// TIA Portal project "Boiler S7 1200+HMI_test_program" (V15)

(* hardware
DEVICE "S7-1200 station_1"  S7-1200 Station
   slot 0: "Rack_0"  S7-1200 Rack  Rack  V1.0
   slot 1: "PLC_BOILER_S71200"  CPU 1214C DC/DC/DC  6ES7 214-1AG40-0XB0  V4.2
   slot 2: "DI 16/DQ 16x24VDC_1"  6ES7 223-1BL32-0XB0  V2.0
   slot 3: "DI 16/DQ 16x24VDC_2"  6ES7 223-1BL32-0XB0  V2.0
   slot 4: "DI 16/DQ 16x24VDC_3"  6ES7 223-1BL32-0XB0  V2.0
   slot 5: "AI 8x13BIT_1"  6ES7 231-4HF32-0XB0  V2.0
   slot 6: "AI 8x13BIT_2"  6ES7 231-4HF32-0XB0  V2.0
   slot 7: "AI 8x13BIT_3"  6ES7 231-4HF32-0XB0  V2.0
   slot 8: "AQ 4x14BIT_1"  6ES7 232-4HD32-0XB0  V2.0
   slot 9: "AQ 4x14BIT_2"  6ES7 232-4HD32-0XB0  V2.0
DEVICE "HMI_BOILER_S71200"  TP1200 Comfort
   slot 0: "HMI_BOILER_S71200"  TP1200 Comfort  6AV2 124-0MC01-0AX0  14.0.1.0
   slot 1: "HMI_RT_2"  TP1200 Comfort  6AV2 124-0MC01-0AX0  14.0.1.0
   slot 5: "HMI_BOILER_S71200.IE_CP_1"  PROFINET Interface  14.0.1.0
      slot 1: "PROFINET Interface_1"  PROFINET Interface
         slot 1: "Port_1"  Port
         slot 2: "Port_2"  Port
   slot 7: "HMI_BOILER_S71200.MPI/DP_CP_1"  MPI/DP Interface  14.0.1.0
*)

// ===== PLC "PLC_BOILER_S71200"  CPU 1214C DC/DC/DC =====

VAR_GLOBAL   // PLC tag table "Default tag table"
   "Tag_2" AT %M4.2 : Bool;
   "Tag_3" AT %M4.3 : Bool;
   "PUMP_COMP_VALUE" AT %MD104 : Real;
   "REFF_PUMPS_FINAL" AT %MD108 : Real;
   "Tag_7" AT %MD128 : Real;
   "Tag_8" AT %MD124 : Real;
   "Tag_9" AT %MD120 : Real;
   "ALRM_Feed_Pump_1_Fault" AT %M15.3 : Bool;
   "ROUND_O2_LEVEL" AT %MD112 : DWord;
   "ROUND SP O2" AT %MD116 : DWord;
   "ID Fan Start" AT %Q0.2 : Bool;
   "Block LH FD Fan" AT %Q4.0 : Bool;
   "Block RH FD Fan" AT %Q4.1 : Bool;
   "Tag_16" AT %M21.5 : Bool;
   "LH_COAL_HEIGHT_0" AT %M13.0 : Bool;
   "RH_COAL_HEIGHT_0" AT %M13.1 : Bool;
   "ALRM_Low_Water_PreWarning" AT %M15.0 : Bool;
   "ALRM_Low_Water" AT %M15.1 : Bool;
   "ALRM_High_Water" AT %M15.2 : Bool;
   "ALRM_Feed_Pump_2_Fault" AT %M15.4 : Bool;
   "ALRM_ID_Fan_Fault" AT %M15.5 : Bool;
   "ALRM_LH_FD_Fan_Fault" AT %M15.6 : Bool;
   "ALRM_RH_FD_Fan_Fault" AT %M15.7 : Bool;
   "ALRM_LH_Stoker_Fault" AT %M14.0 : Bool;
   "ALRM_RH_Stoker_Fault" AT %M14.1 : Bool;
   "ALRM_LH_Swing_Chute_Fault" AT %M14.2 : Bool;
   "ALRM_RH_Swing_Chute_Fault" AT %M14.3 : Bool;
   "ALRM_RAV_1_Fault" AT %M14.4 : Bool;
   "ALRM_RAV_2_Fault" AT %M14.5 : Bool;
   "ALRM_Ash_Conv_Fault" AT %M14.6 : Bool;
   "ALRM_LH_Shearpin_Fault" AT %M14.7 : Bool;
   "ALRM_RH_Shearpin_Fault" AT %M17.0 : Bool;
   "ALRM_LH_Burnback_Fault" AT %M17.1 : Bool;
   "ALRM_RH_Burnback_Fault" AT %M17.2 : Bool;
   "ALRM_Lockout" AT %M17.3 : Bool;
   "ALRM_COAL_Hopper_Low_Level" AT %M17.4 : Bool;
   "ALRM_Steam_Press_Too_Low" AT %M17.5 : Bool;
   "ALRM_Steam_Press_Too_High" AT %M17.6 : Bool;
   "ALRM_EMERGENCY_STOP" AT %M17.7 : Bool;
   "ALRM_Pump_Pressure_Low" AT %M16.1 : Bool;
   "ALRM_Water_Flowrate_Fault" AT %M16.2 : Bool;
   "ALRM_LH_Single_Bucket_Fault" AT %M16.3 : Bool;
   "ALRM_RH_Single_Bucket_Fault" AT %M16.4 : Bool;
   "ALRM_FP_Dry_Run_Protection" AT %M16.5 : Bool;
   "Emergency Stop" AT %I0.0 : Bool;
   "Ready For Operation" AT %I0.1 : Bool;
   "Water Pulser" AT %I0.2 : Bool;
   "Low Water" AT %I0.3 : Bool;
   "Feed Pump 1 Run Status" AT %I0.4 : Bool;
   "Feed Pump 1 VFD Fault" AT %I0.5 : Bool;
   "Feed Pump 2 Run Status" AT %I0.6 : Bool;
   "Feed Pump 2 VFD Fault" AT %I0.7 : Bool;
   "Lock Out" AT %I2.0 : Bool;
   "Pressure Limiter" AT %I2.1 : Bool;
   "Feed Pump 1 SW" AT %I2.2 : Bool;
   "Feed Pump 2 SW" AT %I2.3 : Bool;
   "SW ID" AT %I2.4 : Bool;
   "ID Run" AT %I2.5 : Bool;
   "ID Fault" AT %I2.6 : Bool;
   "SW FD" AT %I2.7 : Bool;
   "LH FD Run" AT %I3.0 : Bool;
   "LH FD Fault" AT %I3.1 : Bool;
   "RH FD Run" AT %I3.2 : Bool;
   "RH FD Fault" AT %I3.3 : Bool;
   "LH Stoker Run" AT %I3.4 : Bool;
   "LH Stoker Fault" AT %I3.5 : Bool;
   "RH Stoker RUN" AT %I3.6 : Bool;
   "RH Stoker Fault" AT %I3.7 : Bool;
   "LH Proximity" AT %I4.0 : Bool;
   "RH Proximity" AT %I4.1 : Bool;
   "LH Swing Chute Run" AT %I4.2 : Bool;
   "CB LH Swing Chute" AT %I4.3 : Bool;
   "RH Swing Chute Run" AT %I4.4 : Bool;
   "CB RH Swing Chute" AT %I4.5 : Bool;
   "Photo No LH" AT %I4.6 : Bool;
   "Photo Nc LH" AT %I4.7 : Bool;
   "ASH Valve 1 Run" AT %I5.0 : Bool;
   "CB ASH Valve 1" AT %I5.1 : Bool;
   "ASH Valve 2 Run" AT %I5.2 : Bool;
   "CB ASH Valve 2" AT %I5.3 : Bool;
   "ASH Conv Run" AT %I5.4 : Bool;
   "VFD Fault ASH Conv" AT %I5.5 : Bool;
   "Horn Off" AT %I5.6 : Bool;
   "Emergency Coal 2" AT %I5.7 : Bool;
   "Bucket 1 Down Status" AT %I6.0 : Bool;
   "Bucket 1 Up Status" AT %I6.1 : Bool;
   "Bucket 2 Up Status" AT %I6.2 : Bool;
   "Coal Empty 1" AT %I6.3 : Bool;
   "Emergency Coal 1" AT %I6.4 : Bool;
   "CB Bucket 1" AT %I6.5 : Bool;
   "Coal Bucket 1 Start Auto" AT %I6.6 : Bool;
   "Bucket 2 Down Status" AT %I6.7 : Bool;
   "Coal 1 Top Limit" AT %I7.0 : Bool;
   "Coal 1 Bottom Limit" AT %I7.1 : Bool;
   "Hand Bucket 1 Down Ext" AT %I7.2 : Bool;
   "Hand Bucket 1 Up Ext" AT %I7.3 : Bool;
   "CB Bucket 2" AT %I7.4 : Bool;
   "Coal Bucket 2 Start Auto" AT %I7.5 : Bool;
   "Coal 2 Top Limit" AT %I7.6 : Bool;
   "Coal 2 Bottom Limit" AT %I7.7 : Bool;
   "Hand Bucket 2 Up Ext" AT %I1.0 : Bool;
   "Dry Run Proximity" AT %I1.1 : Bool;
   "Hand Bucket 2 Down Ext" AT %I1.2 : Bool;
   "Start Feed Pump 1" AT %Q0.0 : Bool;
   "Start Feed Pump 2" AT %Q0.1 : Bool;
   "LH FD Fan Start" AT %Q0.3 : Bool;
   "RH FD Fan Start" AT %Q0.4 : Bool;
   "LH Stoker Start_O" AT %Q0.5 : Bool;
   "RH Stoker Start_O" AT %Q0.6 : Bool;
   "LH Swing" AT %Q0.7 : Bool;
   "RH Swing" AT %Q2.0 : Bool;
   "ASH Valve 1" AT %Q2.1 : Bool;
   "ASH Valve 2" AT %Q2.2 : Bool;
   "ASH Conv" AT %Q2.3 : Bool;
   "Alarm Horn" AT %Q2.4 : Bool;
   "Alarm Flash" AT %Q2.5 : Bool;
   "MPA 26 BLOWDOWN" AT %Q2.6 : Bool;
   "LH Stoker Low" AT %Q2.7 : Bool;
   "RH Stoker Low" AT %Q3.0 : Bool;
   "Coal bucket 1 Up" AT %Q3.1 : Bool;
   "Coal bucket 1 Down" AT %Q3.2 : Bool;
   "Bucket 2 Up" AT %Q3.3 : Bool;
   "ID Fan INC" AT %Q3.4 : Bool;
   "ID Fan Dec" AT %Q3.5 : Bool;
   "Bucket 2 Down" AT %Q3.6 : Bool;
   "Open LH Front Und" AT %Q4.4 : Bool;
   "Close LH Front Und" AT %Q4.5 : Bool;
   "Open RH Front Und" AT %Q4.6 : Bool;
   "Close RH Front Und" AT %Q4.7 : Bool;
   "Open LH Rear Und" AT %Q5.0 : Bool;
   "Close LH Rear Und" AT %Q5.1 : Bool;
   "Open RH Rear Und" AT %Q5.2 : Bool;
   "Close RH Rear Und" AT %Q5.3 : Bool;
   "Water Flow Rate" AT %IW104 : Int;
   "Feed Pump 1 Speed" AT %IW106 : Int;
   "Feed Pump 2 Speed" AT %IW108 : Int;
   "Speed ID Fan" AT %IW110 : Int;
   "Speed LH FD Fan" AT %IW112 : Int;
   "Speed RH FD Fan" AT %IW114 : Int;
   "Tag_142" AT %IW116 : Int;
   "Tag_143" AT %IW118 : Int;
   "Speed LH Stoker" AT %IW200 : Int;
   "Press Transducer" AT %IW100 : Int;
   "Press Pump Line" AT %IW102 : Int;
   "Speed RH Stoker" AT %IW202 : Int;
   "NRGT (Level electrode)" AT %IW204 : Int;
   "O2 Probe" AT %IW206 : Int;
   "Poti LH Front Undergrate" AT %IW208 : Int;
   "Poti RH Front Undergrate" AT %IW212 : Int;
   "Poti LH Rear Undergrate" AT %IW304 : Int;
   "Poti RH Rear Undergrate" AT %IW312 : Int;
   "Water Temp" AT %IW300 : Int;
   "Flue Temp" AT %IW302 : Int;
   "LH Thermocouple" AT %IW308 : Int;
   "RH Thermocouple" AT %IW310 : Int;
   "Feed Pump 1 Reff" AT %QW500 : Int;
   "Feed Pump 2 Reff" AT %QW502 : Int;
   "ID Fan Reff" AT %QW504 : Int;
   "LH FD Fan Reff" AT %QW506 : Int;
   "RH FD Fan Reff" AT %QW600 : Int;
   "LH Stoker Reff" AT %QW602 : Int;
   "RH Stoker Reff" AT %QW604 : Int;
   "Always_True" AT %M1.0 : Bool;
   "Always_False" AT %M1.1 : Bool;
   "Tag_169" AT %M20.3 : Bool;
   "Tag_171" AT %M20.4 : Bool;
   "ALRM_Flash_Command" AT %M11.0 : Bool;
   "Tag_173" AT %M39.2 : Bool;
   "Tag_174" AT %M39.1 : Bool;
   "FORCE STOP PUMPS COMMAND" AT %M0.0 : Bool;
   "Tag_176" AT %M0.1 : Bool;
   "Tag_177" AT %M0.2 : Bool;
   "System_Byte" AT %MB1 : Byte;
   "Tag_m1.2" AT %M1.2 : Bool;
   "Tag_m1.3" AT %M1.3 : Bool;
   "Clock_Byte" AT %MB10 : Byte;
   "Clock_10Hz" AT %M10.0 : Bool;
   "Clock_5Hz" AT %M10.1 : Bool;
   "Clock_2.5Hz" AT %M10.2 : Bool;
   "Clock_2Hz" AT %M10.3 : Bool;
   "Clock_1.25Hz" AT %M10.4 : Bool;
   "Clock_1s" AT %M10.5 : Bool;
   "Clock_0.625Hz" AT %M10.6 : Bool;
   "Clock_0.5Hz" AT %M10.7 : Bool;
   "Tag_1" AT %MD500 : Real;
   "Tag_4" AT %MD504 : Real;
   "Tag_5" AT %MD508 : Real;
END_VAR

DATA_BLOCK "DB1_AREA_POINTER_HMI"   // DB1
{ S7_Optimized_Access := 'FALSE' }
VERSION : 0.1
   VAR
      Coordination : Int;
      Date_Time : Struct
         Write : Struct
            Date_Time : DTL;
            RetVal : Int;
         END_STRUCT;
         Read : Struct
            Date_Time : DTL;
            RetVal : Int;
         END_STRUCT;
         Word_1 : Word;
         Word_2 : Word;
         Word_2_1 : Word;
         Word_2_2 : Word;
         Word_2_3 : Word;
         Word_2_4 : Word;
      END_STRUCT;
      Job_Mail_Box : Struct
         Job_Number : Word;
         Param_1 : Word;
         Param_2 : Word;
         Param_3 : Word;
      END_STRUCT;
      Set_Time : Bool;
      Set_Time_Command : Bool;
   END_VAR
BEGIN
END_DATA_BLOCK

DATA_BLOCK "DB_TEMP_OFFSET"   // DB9
{ S7_Optimized_Access := 'FALSE' }
VERSION : 0.1
   VAR
      LH_BURNBACK_TEMP : Real := 24.93489;
      LH_BURNBACK_OFFSET : Real := 1.0;
      RH_BURNBACK_TEMP : Real := 28.03277;
      RH_BURNBACK_OFFSET : Real := 0.0;
      LH_REAR_UND_POS : Real := 0.0;
      LH_REAR_UND_OFFSET : Real := 0.0;
      RH_REAR_UND_POS : Real := 0.0;
      RH_REAR_UND_OFFSET : Real := 0.0;
      LH_FRONT_UND_POS : Real := 0.0;
      LH_FRONT_UND_OFFSET : Real := 0.0;
      RH_FRONT_UND_POS : Real := 0.0;
      RH_FRONT_UND_OFFSET : Real := 0.0;
   END_VAR
BEGIN
END_DATA_BLOCK

DATA_BLOCK "DB_Scalling"   // DB21
{ S7_Optimized_Access := 'FALSE' }
VERSION : 0.1
   VAR
      Pressurre_Steam_Min : Real;
      Pressure_Steam_Max : Real;
      Pressure_Pump_Min : Real;
      Pressure_Pump_Max : Real;
      Water_Flowrate_Min : Real;
      Water_Flowrate_Max : Real;
      Feed_Pump_1_Min : Real;
      Feed_Pump_1_Max : Real;
      Feed_Pump_2_Min : Real;
      Feed_Pump_2_Max : Real;
      ID_Fan_Min : Real;
      ID_Fan_Max : Real;
      LH_FD_Fan_Min : Real;
      LH_FD_Fan_Max : Real;
      RH_FD_Fan_Min : Real;
      RH_FD_Fan_Max : Real;
      LH_Stoker_Min : Real;
      LH_Stoker_Max : Real;
      RH_Stoker_Min : Real;
      RH_Stoker_Max : Real;
      "NRGT(Water_Level)_Min" : Real;
      "NRGT(Water_Level)_Max" : Real;
      O2_Probe_Min : Real;
      O2_Probe_Max : Real;
      Water_Temp_Min : Real;
      Water_Temp_Max : Real;
      Flue_Min : Real;
      Flue_Max : Real;
      LH_Thermocouple_Min : Real;
      LH_Thermocouple_Max : Real;
      RH_Thermocouple_Min : Real;
      RH_Thermocouple_MAX : Real;
      LH_Front_Undergrate_Min : Real;
      LH_Front_Undergrate_Max : Real;
      RH_Front_Undergrate_Min : Real;
      RH_Front_Undergrate_Max : Real;
      LH_Rear_Undergrate_Min : Real;
      LH_Rear_Undergrate_Max : Real;
      RH_Rear_Undergrate_Min : Real;
      RH_Rear_Undergrate_Max : Real;
      Analog_LH_Front_Min : Real;
      Analog_LH_Front_Max : Real;
      Analog_RH_Front_Min : Real;
      Analog_RH_Front_Max : Real;
      Analog_LH_Rear_Min : Real;
      Analog_LH_Rear_Max : Real;
      Analog_RH_Rear_Min : Real;
      Analog_RH_Rear_Max : Real;
   END_VAR
BEGIN
END_DATA_BLOCK

DATA_BLOCK "DB100_WORK_BIT"   // DB100
{ S7_Optimized_Access := 'FALSE' }
VERSION : 0.1
   VAR
      "STAT0_Start Feed Pump 1" : Bool;
      "STAT1_Start Feed Pump 2" : Bool;
      "STAT2_ID Fan Start" : Bool;
      "STAT3_LH FD Fan Start" : Bool;
      "STAT4_RH FD Fan Start" : Bool;
      "STAT5_LH Stoker Start" : Bool;
      "STAT6_RH Stoker Start" : Bool;
      "STAT7_LH Swing" : Bool;
      "STAT8_RH Swing" : Bool;
      "STAT9_ASH Conv" : Bool;
      STAT10_BUFFTANK1_PUMP_ST : Bool;
      STAT11_BUFFTANK2_PUMP_ST : Bool;
      STAT12_FWT1_PUMP_START : Bool;
      STAT13_FWT2_PUMP_START : Bool;
      STAT14_WETSCRUBBER_PUMP_S : Bool;
      "STAT15_ASH Valve 1 Start" : Bool;
      "STAT16_ASH Valve 2 Start" : Bool;
      "STAT17_Alarm Horn" : Bool;
      "STAT18_Alarm Flash" : Bool;
      "STAT19_MPA 26" : Bool;
      STAT20_DOSING_PUMP1_STAR : Bool;
      STAT21_SUPPLY_VALVE : Bool;
      "STAT22_Water Pulser" : Bool;
      "STAT23_Low Water" : Bool;
      "STAT24_FP 1 Run Status" : Bool;
      "STAT25_FP 2 Run Status" : Bool;
      "STAT26_FP 1 VFD Fault" : Bool;
      "STAT27_FP 2 VFD Fault" : Bool;
      "STAT28_Lock Out" : Bool;
      "STAT29_Pressure Limiter" : Bool;
      "STAT30_ID Run" : Bool;
      "STAT31_LH FD Run" : Bool;
      "STAT32_RH FD Run" : Bool;
      "STAT33_LH Stoker Run" : Bool;
      "STAT34_RH Stoker Run" : Bool;
      "STAT35_LH Stoker Fault" : Bool;
      "STAT36_RH Stoker Fault" : Bool;
      "STAT37_CB LH Swing Chute" : Bool;
      "STAT38_CB RH Swing Chute" : Bool;
      "STAT39_LH Swing Chute Run" : Bool;
      "STAT40_RH Swing Chute Run" : Bool;
      "STAT41_LH Proximity" : Bool;
      "STAT42_RH Proximity" : Bool;
      STAT43_PHOTO_NC : Bool;
      STAT44_PHOTO_NO : Bool;
      "STAT45_CB ASH Valve 1" : Bool;
      "STAT46_CB ASH Valve 2" : Bool;
      "STAT47_VFD Fault ASH Conv" : Bool;
      "STAT48_ASH Conv Run" : Bool;
      STAT49_CB_BUFFTANK1_PUMP : Bool;
      STAT50_CB_BUFFTANK2_PUMP : Bool;
      STAT51_CB_FWT1_PUMP : Bool;
      STAT52_CB_FWT2_PUMP : Bool;
      STAT53_CB_WETSCRUBBER : Bool;
      STAT54_WETSCRUBBER_FB : Bool;
      STAT55_CB_DOSING_PUMP1 : Bool;
      STAT56_SOFTENING_FAULT_I : Bool;
      STAT57_ALWAYS_ON : Bool := TRUE;
      STAT58_PUMPS_ON : Bool;
      STAT59_PUMPS_OFF : Bool;
      STAT60_DRY_RUN_PROTECTIO : Bool;
      STAT61_FORCE_PUMPS_STOP : Bool;
      STAT62_NW_INPUT : Bool;
      "STAT63_ID Fault" : Bool;
      "STAT64_LH FD Fault" : Bool;
      "STAT65_RH FD Fault" : Bool;
      "STAT66_Ready For Operation" : Bool;
      STAT67_Ready : Bool;
      "STAT68_LH Stoker Low" : Bool;
      "STAT69_RH Stoker Low" : Bool;
      STAT70WASTE_WATER_PUMP_S : Bool;
      STAT71_CB_WW_PUMP : Bool;
      "STAT72_ASH Valve 1 Run" : Bool;
      "STAT73_ASH Valve 2 Run" : Bool;
      STAT74_CB_DOSING_PUMP2 : Bool;
      STAT75_DOSING_PUMP2_STAR : Bool;
      STAT76_CB_COAL_CONV1 : Bool;
      STAT77_CB_COAL_CONV2 : Bool;
      STAT78_COAL_CONV1_START : Bool;
      STAT79_COAL_CONV2_START : Bool;
      STAT80_CB_RAV3 : Bool;
      STAT81_RAV3_START : Bool;
      STAT82_ON_DELAY_SINGLE_B : Time;
      STAT83_HAND_0PEN_ECO : Bool;
      STAT84_ECO_OPEN : Bool;
      STAT85_ECO_CLOSE : Bool;
      STAT86_COAL_CONV1_FB : Bool;
      STAT87_COAL_CONV2_FB : Bool;
      STAT88_RAV3_FB : Bool;
      "STAT89_ID Fan INC" : Bool;
      "STAT90_ID Fan Dec" : Bool;
      "STAT91_Bucket 1 Down Status" : Bool;
      "STAT92_Bucket 1 Up Status" : Bool;
      "STAT93_Bucket 2 Up Status" : Bool;
      STAT94_EMG_LH_BUCKET : Bool;
      STAT95_EMG_RH_BUCKET : Bool;
      "STAT96_CB Bucket 1" : Bool;
      "STAT97_CB Bucket 2" : Bool;
      STAT98_LH_BUCKET_START_A : Bool;
      "STAT99_Bucket 2 Down Status" : Bool;
      STAT100_LH_TOP_LIMIT : Bool;
      STAT101_LH_BOTTOM_LIMIT : Bool;
      STAT102_RH_TOP_LIMIT : Bool;
      STAT103_RH_BOTTOM_LIMIT : Bool;
      STAT104_RH_BUCKET_START_A : Bool;
      STAT105_HAND_LH_BUCKET_U : Bool;
      STAT106_HAND_LH_BUCKET_D : Bool;
      STAT107_HAND_RH_BUCKET_U : Bool;
      STAT108_HAND_RH_BUCKET_D : Bool;
      STAT109_LH_SINGLE_BUCKET_UP : Bool;
      STAT110_LH_SINGLE_BUCKET_DOWN : Bool;
      STAT111_RH_SINGLE_BUCKET_UP : Bool;
      STAT112_RH_SINGLE_BUCKET_DOWN : Bool;
      "STAT113_Open LH Front Und" : Bool;
      "STAT114_Close LH Front Und" : Bool;
      "STAT115_Open RH Front Und" : Bool;
      "STAT116_Close RH Front Und" : Bool;
      "STAT117_Open LH Rear Und" : Bool;
      "STAT118_Close LH Rear Und" : Bool;
      "STAT119_Open RH Rear Und" : Bool;
      "STAT120_Close RH Rear Und" : Bool;
   END_VAR
BEGIN
END_DATA_BLOCK

DATA_BLOCK "DB101_DATA_SWITCH"   // DB101
{ S7_Optimized_Access := 'FALSE' }
VERSION : 0.1
   VAR
      STAT0_AUTO_FP : Bool := false;
      STAT1_FEED_PUMP_1_SW : Bool;
      STAT2_FEED_PUMP_2_SW : Bool;
      "STAT3_SW ID" : Bool;
      "STAT4_SW FD" : Bool;
      STAT5_SW_LHSTOKER : Bool;
      STAT6_SW_RHSTOKER : Bool;
      STAT7_SW_ASH_CONV : Bool;
      STAT8_SW_LHSWING : Bool;
      STAT9_SW_RHSWING : Bool;
      STAT10_AUTO_ID : Bool;
      STAT11_AUTO_LHFD : Bool;
      STAT12_AUTO_LHSTOKER : Bool;
      STAT13_AUTO_RHSTOKER : Bool;
      STAT14_AUTO_LHSWING : Bool;
      STAT15_AUTO_RHSWING : Bool;
      "STAT16_Emergency Stop" : Bool;
      STAT17_EMG_MCC : Bool;
      STAT18_FWT_FILLING_SW : Bool;
      STAT19_FWT_BLANK_SW : Bool;
      STAT20_FWT_BRIMFULL_SW : Bool;
      STAT21_BFTANK_FILLING_SW : Bool;
      STAT22_BFTANK_BLANK_SW : Bool;
      STAT23_BFTANK_BRIMFULL_S : Bool;
      STAT24_SW_WETSCRUBBER : Bool;
      STAT25_HAND_SPEED_UP_ID : Bool;
      STAT26_HAND_SPEED_DOWN_I : Bool;
      STAT27_HAND_SPEED_UP_LHF : Bool;
      STAT28_HAND_SPEED_DOWN_L : Bool;
      STAT29_HAND_SPEED_UP_RHF : Bool;
      STAT30_HAND_SPEED_DOWN_R : Bool;
      STAT31_HAND_SPEED_UP_LHS : Bool;
      STAT32_HAND_SPEED_DOWN_L : Bool;
      STAT33_HAND_SPEED_UP_RHS : Bool;
      STAT34_HAND_SPEED_DOWN_R : Bool;
      STAT35_SW_BUFTANK_PUMP1 : Bool;
      STAT36_SW_BUFTANK_PUMP2 : Bool;
      STAT37_SW_FWT_PUMP1 : Bool;
      STAT38_SW_FWT_PUMP2 : Bool;
      STAT39_SW_WWT_PUMP : Bool;
      STAT40_SW_DOSING1 : Bool;
      STAT41_AUTO_LHFRONT_UND_S : Bool;
      STAT42_AUTO_RHFRONT_UND_S : Bool;
      "STAT43_Horn Off" : Bool;
      "STAT44_Coal Empty 1" : Bool;
      STAT45_AUTO_BUFF_PUMP : Bool;
      STAT46_AUTO_FWTANK_PUMP : Bool;
      STAT47_AUTO_DOSING_PUMP1 : Bool;
      STAT48_AUTO_DOSING_PUMP2 : Bool;
      STAT49_HAND_DOSING1_SW : Bool;
      STAT50_HAND_DOSING2_SW : Bool;
      STAT51_AUTO_RHFD : Bool;
      STAT52_SW_DOSING2 : Bool;
      STAT53_LH_HAND_BUCKET_UP : Bool;
      STAT54_LH_HAND_BUCKET_DO : Bool;
      STAT55_RH_HAND_BUCKET_DO : Bool;
      STAT56_AUTO_LH_BUCKET : Bool;
      STAT57_AUTO_RH_BUCKET : Bool;
      STAT58_COAL_CONV1_SW_HMI : Bool;
      STAT59_COAL_CONV1_SW_LOC : Bool;
      "STAT60_Dry Run Proximity" : Bool;
      "STAT61_Emergency Coal 2" : Bool;
      STAT62_COAL_CONV2_SW_HMI : Bool;
      STAT63_COAL_CONV2_SW_LOC : Bool;
      "STAT64_Coal 2 Top Limit" : Bool;
      "STAT65_Coal 2 Bottom Limit" : Bool;
      "STAT66_Hand Bucket 1 Down Ext" : Bool;
      "STAT67_Hand Bucket 1 Up Ext" : Bool;
      "STAT68_Hand Bucket 2 Up Ext" : Bool;
      "STAT69_Hand Bucket 2 Down Ext" : Bool;
      STAT70_RH_HAND_BUCKET_UP : Bool;
      STAT71_AUTO_ECO : Bool;
      STAT72_HAND_OPEN_ECO : Bool;
      STAT73_HAND_CLOSE_ECO : Bool;
      STAT74_ECO_WATER_LIMITER : Bool;
      "STAT75_Coal 1 Top Limit" : Bool;
      "STAT76_Coal 1 Bottom Limit" : Bool;
      "STAT77_Coal Bucket 1 Start Auto" : Bool;
      "STAT78_Coal Bucket 2 Start Auto" : Bool;
      STAT79_HAND_LH_FRONT_UND_O : Bool;
      STAT80_HAND_LH_FRONT_UND_C : Bool;
      STAT81_HAND_RH_FRONT_UND_O : Bool;
      STAT82_HAND_RH_FRONT_UND_C : Bool;
      STAT83_O2_CONTROL_ENABLE : Bool;
      STAT84_HAND_LH_REAR_UND_O : Bool;
      STAT85_HAND_LH_REAR_UND_C : Bool;
      STAT86_HAND_RH_REAR_UND_O : Bool;
      STAT87_HAND_RH_REAR_UND_C : Bool;
      STAT88_HAND_SPEED_UP_FP : Bool;
      STAT89_HAND_SPEED_DOWN_F : Bool;
      STAT90_HAND_AUTO_BLOWDOWN : Bool;
      STAT91_PB_BLOWDOWN : Bool;
   END_VAR
BEGIN
END_DATA_BLOCK

DATA_BLOCK "DB102_ANALOG_DISPLAY"   // DB102
{ S7_Optimized_Access := 'FALSE' }
VERSION : 0.1
   VAR
      STAT0_WATER_LEVEL : Real;
      STAT1_STEAM_PRESSURE : Real;
      STAT2_PUMP_PRESSURE : Real;
      STAT3_WATER_FLOWRATE : Real;
      STAT4_STEAM_FLOW_NEW_BOI : Real;
      STAT5_FP1_SPEED : Real;
      STAT6_FP2_SPEED : Real;
      STAT7_ID_SPEED : Real;
      STAT8_LHFD_SPEED : Real;
      STAT9_RHFD_SPEED : Real;
      STAT10_LHSTOKER_SPEED : Real;
      STAT11_RHSTOKER_SPEED : Real;
      STAT12_O2_LEVEL : Real;
      STAT13_CO2_LEVEL : Real;
      STAT14_WATER_TEMP : Real;
      STAT15_FLUE_GAS_TEMP : Real;
      STAT16_LH_BURNBACK_TEMP : Real;
      STAT17_RH_BURNBACK_TEMP : Real;
      STAT18_LH_FRONT_UND_POS : Real;
      STAT19_RH_FRONT_UND_POS : Real;
      STAT20_LH_REAR_UND_POS : Real;
      STAT21_RH_REAR_UND_POS : Real;
      STAT22_STEAM_FLOW_DEAERA : Real;
      STAT23_STEAM_FLOW_OLDBOI : Real;
      STAT24_TOTAL_WATER : Real;
      STAT25_LH_TOTAL_COAL : Real;
      STAT26_RH_TOTAL_COAL : Real;
      STAT27_WATER_TEMP_ECO : Real;
      STAT28 : Real;
      STAT29 : Real;
   END_VAR
BEGIN
END_DATA_BLOCK

DATA_BLOCK "DB103_ANALOG_INPUT"   // DB103
{ S7_Optimized_Access := 'FALSE' }
VERSION : 0.1
   VAR
      "STAT0_NRGT (Level electrode)" : Int;
      "STAT1_Press Transducer" : Int;
      "STAT2_Press Pump Line" : Int;
      "STAT3_Water Temp" : Int;
      "STAT4_Flue Temp" : Int;
      "STAT5_LH Thermocouple" : Int;
      "STAT6_RH Thermocouple" : Int;
      "STAT7_Feed Pump 1 Speed" : Int;
      "STAT8_Feed Pump 2 Speed" : Int;
      "STAT9_Speed ID Fan" : Int;
      STAT10_AOC_FD : Int;
      "STAT11_Speed LH FD Fan" : Int;
      "STAT12_Speed RH FD Fan" : Int;
      "STAT13_Speed LH Stoker" : Int;
      "STAT14_Speed RH Stoker" : Int;
      "STAT15_Poti LH Front Undgrt" : Int;
      "STAT16_Poti RH Front Undgrt" : Int;
      "STAT17_Poti LH Rear Undgrt" : Int;
      "STAT18_Poti RH Rear Undgrt" : Int;
      STAT19_STEAM_FLOW_BOILER : Int;
      STAT20_STEAM_FLOW_DEAERA : Int;
      STAT21_STEAM_FLOW_OLDBOI : Int;
      "STAT22_O2 Probe" : Int;
      "STAT23_Water Flow Rate" : Int;
      STAT24_PT_100_ECO : Int;
      STAT25 : Int;
      STAT26 : Int;
   END_VAR
BEGIN
END_DATA_BLOCK

DATA_BLOCK "DB104_WTR_LEVEL_SCALING"   // DB104
{ S7_Optimized_Access := 'TRUE' }
VERSION : 0.1
// stored: InstanceOfName FB20_RA_AI
"FB20_RA_AI"
BEGIN
   IN4 := 100.0;
   IN5 := 5.0;
   IN6 := 25.0;
   IN7 := 80.0;
   IN8 := 100.0;
END_DATA_BLOCK

DATA_BLOCK "DB106_DATA_PARAMETER"   // DB106
{ S7_Optimized_Access := 'FALSE' }
VERSION : 0.1
   VAR
      STAT0_SP_WATER_LEVEL : Real := 65.0;
      STAT1_SP_FD : Real := 0.0;
      STAT2 : Real := 0.0;
      STAT3 : Real := 0.0;
      STAT4_HAND_REFF_FP : Real := 100.0;
      STAT5_MAX_FLOWRATE : Real := 27.0;
      STAT6 : Real := 0.0;
      STAT7 : Real := 0.0;
      STAT8 : Real := 0.0;
      STAT9 : Real := 0.0;
      STAT10 : Real := 0.0;
      STAT11_AUTO_MIN_WATER_LEVEL : Real := 60.0;
      STAT12_IDFAN_SPEED_REFF : Real := 96.0;
      STAT13_HAND_REFF_LHFD_FA : Real := 46.0;
      STAT14_HAND_REFF_RHFD_FA : Real := 58.5;
      STAT15 : Real;
      STAT16 : Real;
      STAT17_LSP_ID_FAN : Real := 48.0;
      STAT18_OUT_PID_FD : Real := 50.0;
      STAT19_PID_OUT_FD : Real := 50.0;
      STAT20_LSP_LHFD_FAN : Real := 20.0;
      STAT21_HSP_LHFD_FAN : Real := 26.0;
      STAT22_LSP_LH_STOKER : Real := 30.0;
      STAT23_HSP_LH_STOKER : Real := 40.0;
      STAT24_PID_OUT_STOKER : Real := 50.0;
      STAT25_LH_OFFSET : DInt := L#50;
      STAT26_RH_OFFSET : DInt := L#50;
      STAT27 : Real;
      STAT28 : Real;
      STAT29 : Real;
      STAT30 : Real;
      STAT31 : Real;
      STAT32 : Real;
      STAT33 : Real;
      STAT34 : Real;
      STAT35 : Real;
      STAT36 : Real;
      STAT37 : Real;
      STAT38 : Real;
      STAT39_LH_COAL_HEIGHT : Real := 150.0;
      STAT40_RH_COAL_HEIGHT : Real := 150.0;
      STAT41_LH_DENSITY : Real := 0.773;
      STAT42_RH_DENSITY : Real := 0.773;
      STAT43 : Real;
      STAT44_OFF_PULSE_BLOWDOW : Time := T#10s;
      STAT45_ON_PULSE_BLOWDOWN : Time := T#10s;
      STAT46_PERIODE_BLOWDOWN : Int := 3;
      STAT47_LSP_PUMP_PERCENT : Real := 80.0;
      STAT48 : Real;
      STAT49 : Real;
      STAT50 : Real;
      STAT51 : Real;
      STAT52_LSP_RHFD_FAN : Real := 20.0;
      STAT53_HSP_RHFD_FAN : Real := 25.0;
      STAT54_MIN_RAW_LHFD : Real := 11059.0;
      STAT55_MAX_RAW_LHFD : Real := 14376.0;
      STAT56 : Real;
      STAT57 : Real;
      STAT58_HAND_REFF_LH_STOK : Real := 35.0;
      STAT59_HAND_REFF_RH_STOK : Real := 35.0;
      STAT60_LSP_RH_STOKER : Real := 30.0;
      STAT61_HSP_RH_STOKER : Real := 40.0;
      STAT62_MIN_RAW_RHFD : Real := 11059.0;
      STAT63_MAX_RAW_RHFD : Real := 13824.0;
      STAT64_MIN_RAW_LH_STOKER : Real := 16588.0;
      STAT65_MAX_RAW_LH_STOKER : Real := 22118.0;
      STAT66_MIN_RAW_RH_STOKER : Real := 16588.0;
      STAT67_MAX_RAW_RH_STOKER : Real := 22118.0;
      STAT68_DELAY_TIME_LH_BUC : Time := T#7s;
      STAT69_DELAY_TIME_RH_BUC : Time := T#7s;
      STAT70_SP_LH_FRONT_UND : DInt := L#0;
      STAT71_SP_RH_FRONT_UND : DInt := L#0;
      STAT72_LH_FRONT_UND_POS_R : DInt := L#-4;
      STAT73_RH_FRONT_UND_POS_R : DInt := L#-7;
      STAT74 : Time := T#3m;
      STAT75_PID_FD_ROUND : DInt := L#50;
      STAT76 : DInt := L#0;
      STAT77_SP_O2 : Real := 3.5;
      STAT78_AUTO_REFF_FD : Real := 50.0;
      STAT79_O2_COMPENSATE_VAL : Real := 4.5;
      STAT80 : Time := T#5m;
      FP_GAIN : Real := 0.2;
      FP_I : Real := 25.0;
      FP_TD : Real := 0.45;
      STAT84_OUT_PID_PUMP : Real := 100.0;
      STAT85_LSP_PUMPS : Real := 40.0;
      STAT86_AUTO_MAX_WATER_LEVEL : Real := 80.0;
      STAT87_OFF_TIME_BLOWDOWN : Int := 480;
   END_VAR
BEGIN
END_DATA_BLOCK

DATA_BLOCK "DB107_SPEED_REF_FP1"   // DB107
{ S7_Optimized_Access := 'TRUE' }
VERSION : 0.1
// stored: InstanceOfName FB21_RA_AO
"FB21_RA_AO"
BEGIN
   IN4 := 100.0;
   IN5 := 5.0;
   IN6 := 15.0;
   IN7 := 85.0;
   IN8 := 95.0;
END_DATA_BLOCK

DATA_BLOCK "DB108_FP_PRESSURE"   // DB108
{ S7_Optimized_Access := 'TRUE' }
VERSION : 0.1
// stored: InstanceOfName FB20_RA_AI
"FB20_RA_AI"
BEGIN
   IN4 := 25.0;
   IN5 := 5.0;
   IN6 := 15.0;
   IN7 := 85.0;
   IN8 := 95.0;
END_DATA_BLOCK

DATA_BLOCK "DB109_STEAM_PRESS"   // DB109
{ S7_Optimized_Access := 'TRUE' }
VERSION : 0.1
// stored: InstanceOfName FB20_RA_AI
"FB20_RA_AI"
BEGIN
   IN4 := 25.0;
   IN5 := 5.0;
   IN6 := 8.5;
   IN7 := 11.5;
   IN8 := 95.0;
END_DATA_BLOCK

DATA_BLOCK "DB110_HZ_TO_PERCENT_LSP_FP"   // DB110
{ S7_Optimized_Access := 'TRUE' }
VERSION : 0.1
// stored: InstanceOfName FB1_HZ_TO_PERCENT
"FB1_HZ_TO_PERCENT"
BEGIN
   IN0 := 40.0;
   IN1 := 50.0;
   Out2 := 80.0;
   STAT3 := 0.8;
END_DATA_BLOCK

DATA_BLOCK "DB115_SPEED_REF_FP2"   // DB115
{ S7_Optimized_Access := 'TRUE' }
VERSION : 0.1
// stored: InstanceOfName FB21_RA_AO
"FB21_RA_AO"
BEGIN
   IN4 := 100.0;
   IN5 := 5.0;
   IN6 := 15.0;
   IN7 := 85.0;
   IN8 := 95.0;
   IN3 := 100.0;
   Out13 := 27648;
   IO19 := 100.0;
END_DATA_BLOCK

DATA_BLOCK "DB116_FEED PUMPS VSD 1 SPEED D"   // DB116
{ S7_Optimized_Access := 'TRUE' }
VERSION : 0.1
// stored: InstanceOfName FB20_RA_AI
"FB20_RA_AI"
BEGIN
   IN4 := 50.0;
   IN5 := 5.0;
   IN6 := 15.0;
   IN7 := 85.0;
   IN8 := 95.0;
END_DATA_BLOCK

DATA_BLOCK "DB117_FEED PUMP VSD 2 SPEED DI"   // DB117
{ S7_Optimized_Access := 'TRUE' }
VERSION : 0.1
// stored: InstanceOfName FB20_RA_AI
"FB20_RA_AI"
BEGIN
   IN4 := 50.0;
   IN5 := 5.0;
   IN6 := 15.0;
   IN7 := 85.0;
   IN8 := 95.0;
END_DATA_BLOCK

DATA_BLOCK "DB120_TEMP_DATA"   // DB120
{ S7_Optimized_Access := 'FALSE' }
VERSION : 0.1
   VAR
      STAT0 : Real;
      STAT1 : Real;
      STAT2 : Real;
      STAT3 : Real;
      STAT4_PUMPS_AUTO_COMMAND : Bool := 0;
      STAT5 : Real;
      STAT6_IDFAN_LSP_PERCENT : Real := 96.0;
      STAT7_FDFAN_PID_OUT_PERCENT : Real := 100.0;
      STAT8 : Real;
      STAT9 : Real;
      STAT10 : Real;
      STAT11 : Real;
      STAT12_ROUND_SCALE_LH_SPEED : DInt := L#0;
      STAT13 : DInt := L#0;
      STAT14 : Real;
      STAT15_ROUND_SCALLING_RH_FD_OUT : DInt := L#0;
      STAT16 : DInt := L#0;
      STAT17 : Real;
      STAT18_LOW_WATER_PREWARN_HORN_OFF : Bool;
      STAT19_LOW_WATER_HORN_OFF : Bool;
      STAT20_HIGH_WATER_HORN_OFF : Bool;
      STAT21_FP1_FAULT_HORN_OFF : Bool;
      STAT22_FP2_FAULT_HORN_OFF : Bool;
      STAT23_ID_FAN_FAULT_HORN_OFF : Bool;
      STAT24_LH_FD_FAULT_HORN_OFF : Bool;
      STAT25_RH_FD_FAULT_HORN_OFF : Bool;
      STAT26_LH_STOKER_FAULT_HORN_OFF : Bool;
      STAT27_RH_STOKER_FAULT_HORN_OFF : Bool;
      STAT28_LH_SWING_FAULT_HORN_OFF : Bool;
      STAT29_RH_SWING_FAULT_HORN_OFF : Bool;
      STAT30_AV1_FAULT_HORN_OFF : Bool;
      STAT31_AV2_FAULT_HORN_OFF : Bool;
      STAT32_ASH_CONV_FAULT_HORN_OFF : Bool;
      STAT33_LH_SHEARPIN_FAULT_HORN_OFF : Bool;
      STAT34_RH_SHEARPIN_FAULT_HORN_OFF : Bool;
      STAT35_LH_BURNBACK_FAULT_HORN_OFF : Bool;
      STAT36_RH_BURNBACK_FAULT_HORN_OFF : Bool;
      STAT37_LOCKOUT_HORN_OFF : Bool;
      STAT38_HOPPER_LL_HORN_OFF : Bool;
      STAT39_STEAM_TO_LOW_HORN_OFF : Bool;
      STAT40_STEAM_TO_HIGH_HORN_OFF : Bool;
      STAT41_EMC_HORN_OFF : Bool;
      STAT42 : Bool;
      STAT43 : Bool;
      STAT44 : Bool;
      STAT45 : Bool;
      STAT46 : Bool;
      STAT47 : Bool;
      STAT48 : Bool;
      STAT49 : Bool;
      STAT50 : Bool;
      STAT51 : Bool;
      STAT52 : Bool;
      STAT53_PUMP_PRESS_LOW_HORN_OFF : Bool;
      STAT54_WATER_FLOWRATE_FAULT_HORN_OFF : Bool;
      STAT55 : Bool;
      STAT56 : Bool;
      STAT57 : Bool;
      STAT58 : Bool;
      STAT59 : Bool;
      STAT60 : Bool;
      STAT61 : Bool;
      STAT62_LH_SB_FAULT_HORN_OFF : Bool;
      STAT63_RH_SB_FAULT_HORN_OFF : Bool;
      STAT64_DRY_RUN_PROTECT_HORN_OFF : Bool;
      STAT65 : Int := 11059;
      STAT66 : Int := 14376;
      STAT67 : DInt := L#11059;
      STAT68 : DInt := L#14376;
      STAT69 : Int := 11059;
      STAT70 : Int := 13824;
      STAT71 : DInt := L#11059;
      STAT72 : DInt := L#13824;
      STAT73 : Int := 16588;
      STAT74 : Int := 22118;
      STAT75 : Int := 16588;
      STAT76 : Int := 22118;
      STAT77 : DInt := L#16588;
      STAT78 : DInt := L#22188;
      STAT79 : DInt := L#16588;
      STAT80 : DInt := L#22188;
   END_VAR
BEGIN
END_DATA_BLOCK

DATA_BLOCK "DB121_ID_FAN_SPEED"   // DB121
{ S7_Optimized_Access := 'TRUE' }
VERSION : 0.1
// stored: InstanceOfName FB20_RA_AI
"FB20_RA_AI"
BEGIN
   IN4 := 50.0;
   IN5 := 5.0;
   IN6 := 15.0;
   IN7 := 85.0;
   IN8 := 95.0;
END_DATA_BLOCK

DATA_BLOCK "DB122_LHFD_SPEED"   // DB122
{ S7_Optimized_Access := 'TRUE' }
VERSION : 0.1
// stored: InstanceOfName FB20_RA_AI
"FB20_RA_AI"
BEGIN
   IN4 := 50.0;
   IN5 := 5.0;
   IN6 := 15.0;
   IN7 := 85.0;
   IN8 := 95.0;
END_DATA_BLOCK

DATA_BLOCK "DB123_RHFD_SPEED"   // DB123
{ S7_Optimized_Access := 'TRUE' }
VERSION : 0.1
// stored: InstanceOfName FB20_RA_AI
"FB20_RA_AI"
BEGIN
   IN4 := 50.0;
   IN5 := 5.0;
   IN6 := 15.0;
   IN7 := 85.0;
   IN8 := 95.0;
END_DATA_BLOCK

DATA_BLOCK "DB124_LH_STOKER_SPEED"   // DB124
{ S7_Optimized_Access := 'TRUE' }
VERSION : 0.1
// stored: InstanceOfName FB20_RA_AI
"FB20_RA_AI"
BEGIN
   IN4 := 50.0;
   IN5 := 5.0;
   IN6 := 15.0;
   IN7 := 85.0;
   IN8 := 95.0;
END_DATA_BLOCK

DATA_BLOCK "DB125_RH_STOKER_SPEED"   // DB125
{ S7_Optimized_Access := 'TRUE' }
VERSION : 0.1
// stored: InstanceOfName FB20_RA_AI
"FB20_RA_AI"
BEGIN
   IN4 := 50.0;
   IN5 := 5.0;
   IN6 := 15.0;
   IN7 := 85.0;
   IN8 := 95.0;
END_DATA_BLOCK

DATA_BLOCK "DB126_O2_LEVEL"   // DB126
{ S7_Optimized_Access := 'TRUE' }
VERSION : 0.1
// stored: InstanceOfName FB20_RA_AI
"FB20_RA_AI"
BEGIN
   IN4 := 20.9;
   IN5 := 5.0;
   IN6 := 15.0;
   IN7 := 85.0;
   IN8 := 95.0;
END_DATA_BLOCK

DATA_BLOCK "DB127_FLUE_GAS_TEMP"   // DB127
{ S7_Optimized_Access := 'TRUE' }
VERSION : 0.1
// stored: InstanceOfName FB20_RA_AI
"FB20_RA_AI"
BEGIN
   IN4 := 400.0;
   IN5 := 5.0;
   IN6 := 15.0;
   IN7 := 85.0;
   IN8 := 95.0;
END_DATA_BLOCK

DATA_BLOCK "DB128_WTR_TEMP"   // DB128
{ S7_Optimized_Access := 'TRUE' }
VERSION : 0.1
// stored: InstanceOfName FB20_RA_AI
"FB20_RA_AI"
BEGIN
   IN4 := 400.0;
   IN5 := 5.0;
   IN6 := 15.0;
   IN7 := 85.0;
   IN8 := 95.0;
END_DATA_BLOCK

DATA_BLOCK "DB129_LH_BURNBACK_TEMP"   // DB129
{ S7_Optimized_Access := 'TRUE' }
VERSION : 0.1
// stored: InstanceOfName FB20_RA_AI
"FB20_RA_AI"
BEGIN
   IN4 := 2764.8;
   IN5 := 5.0;
   IN6 := 15.0;
   IN7 := 999.0;
   IN8 := 95.0;
END_DATA_BLOCK

DATA_BLOCK "DB130_RH_BURNBACK_TEMP"   // DB130
{ S7_Optimized_Access := 'TRUE' }
VERSION : 0.1
// stored: InstanceOfName FB20_RA_AI
"FB20_RA_AI"
BEGIN
   IN4 := 2764.8;
   IN5 := 5.0;
   IN6 := 15.0;
   IN7 := 999.0;
   IN8 := 95.0;
END_DATA_BLOCK

DATA_BLOCK "DB131_LH_FRONT_UND"   // DB131
{ S7_Optimized_Access := 'TRUE' }
VERSION : 0.1
// stored: InstanceOfName FB23_RA_AI_CUSTOM
"FB23_RA_AI_CUSTOM"
BEGIN
   IN5 := 5.0;
   IN6 := 15.0;
   IN7 := 85.0;
   IN8 := 95.0;
END_DATA_BLOCK

DATA_BLOCK "DB132_RH_FRONT_UND"   // DB132
{ S7_Optimized_Access := 'TRUE' }
VERSION : 0.1
// stored: InstanceOfName FB23_RA_AI_CUSTOM
"FB23_RA_AI_CUSTOM"
BEGIN
   IN5 := 5.0;
   IN6 := 15.0;
   IN7 := 85.0;
   IN8 := 95.0;
END_DATA_BLOCK

DATA_BLOCK "DB133_LH_REAR_UND"   // DB133
{ S7_Optimized_Access := 'TRUE' }
VERSION : 0.1
// stored: InstanceOfName FB23_RA_AI_CUSTOM
"FB23_RA_AI_CUSTOM"
BEGIN
   IN5 := 5.0;
   IN6 := 15.0;
   IN7 := 85.0;
   IN8 := 95.0;
END_DATA_BLOCK

DATA_BLOCK "DB134_RH_REAR_UND"   // DB134
{ S7_Optimized_Access := 'TRUE' }
VERSION : 0.1
// stored: InstanceOfName FB23_RA_AI_CUSTOM
"FB23_RA_AI_CUSTOM"
BEGIN
   IN5 := 5.0;
   IN6 := 15.0;
   IN7 := 85.0;
   IN8 := 95.0;
END_DATA_BLOCK

DATA_BLOCK "DB138_HZ_TO_PERCENT_LSP_IDFAN"   // DB138
{ S7_Optimized_Access := 'TRUE' }
VERSION : 0.1
// stored: InstanceOfName FB1_HZ_TO_PERCENT
"FB1_HZ_TO_PERCENT"
BEGIN
   IN0 := 48.0;
   IN1 := 50.0;
   Out2 := 96.0;
   STAT3 := 0.96;
END_DATA_BLOCK

DATA_BLOCK "DB139_HZ_TO_PERCENT_OUT_PID_FDFAN"   // DB139
{ S7_Optimized_Access := 'TRUE' }
VERSION : 0.1
// stored: InstanceOfName FB1_HZ_TO_PERCENT
"FB1_HZ_TO_PERCENT"
BEGIN
   IN0 := 50.0;
   IN1 := 50.0;
   Out2 := 100.0;
   STAT3 := 1.0;
END_DATA_BLOCK

DATA_BLOCK "DB140_ANALOG_OUTPUT"   // DB140
{ S7_Optimized_Access := 'FALSE' }
VERSION : 0.1
   VAR
      "STAT0_ID Fan Reff" : Int := 26542;
      "STAT1_Speed LH FD Reff" : Int := 14110;
      "STAT2_RH FD Fan Reff" : Int := 13824;
      "STAT3_LH Stoker Reff" : Int := 22118;
      "STAT4_RH Stoker Reff" : Int := 22118;
      STAT5LH_FRONT_UND_REFF_O : Int;
      STAT6RH_FRONT_UND_REFF_O : Int;
      STAT7_LH_REAR_UND_REFF_O : Int;
      STAT8_RH_REAR_UND_REFF_O : Int;
      "STAT9_Feed Pump 1 Reff" : Int := 27648;
      "STAT10_Feed Pump 2 Reff" : Int := 27648;
      STAT11_ASH_CONV_REFF_OUT : Int;
   END_VAR
BEGIN
END_DATA_BLOCK

DATA_BLOCK "DB141_ID_FAN_REFF_OUT"   // DB141
{ S7_Optimized_Access := 'TRUE' }
VERSION : 0.1
// stored: InstanceOfName FB21_RA_AO
"FB21_RA_AO"
BEGIN
   IN4 := 50.0;
   IN5 := 5.0;
   IN6 := 15.0;
   IN7 := 85.0;
   IN8 := 95.0;
   IN3 := 50.0;
END_DATA_BLOCK

DATA_BLOCK "DB143_LHFD_REF_OUT"   // DB143
{ S7_Optimized_Access := 'TRUE' }
VERSION : 0.1
// stored: InstanceOfName FB22_RA_AO_CUSTOM
"FB22_RA_AO_CUSTOM"
BEGIN
   IN4 := 100.0;
   IN5 := 5.0;
   IN6 := 15.0;
   IN7 := 85.0;
   IN8 := 95.0;
END_DATA_BLOCK

DATA_BLOCK "DB144_RHFD_SPEED_REF"   // DB144
{ S7_Optimized_Access := 'TRUE' }
VERSION : 0.1
// stored: InstanceOfName FB22_RA_AO_CUSTOM
"FB22_RA_AO_CUSTOM"
BEGIN
   IN4 := 100.0;
   IN5 := 5.0;
   IN6 := 15.0;
   IN7 := 85.0;
   IN8 := 95.0;
END_DATA_BLOCK

DATA_BLOCK "DB148_LH_STOKER_REFF_OUT"   // DB148
{ S7_Optimized_Access := 'TRUE' }
VERSION : 0.1
// stored: InstanceOfName FB21_RA_AO
"FB21_RA_AO"
BEGIN
   IN4 := 100.0;
   IN5 := 5.0;
   IN6 := 15.0;
   IN7 := 85.0;
   IN8 := 95.0;
END_DATA_BLOCK

DATA_BLOCK "DB149_RH_STOKER_REFF_OUT"   // DB149
{ S7_Optimized_Access := 'TRUE' }
VERSION : 0.1
// stored: InstanceOfName FB21_RA_AO
"FB21_RA_AO"
BEGIN
   IN4 := 100.0;
   IN5 := 5.0;
   IN6 := 15.0;
   IN7 := 85.0;
   IN8 := 95.0;
END_DATA_BLOCK

DATA_BLOCK "DB152_WATER_FLOWRATE"   // DB152
{ S7_Optimized_Access := 'TRUE' }
VERSION : 0.1
// stored: InstanceOfName FB20_RA_AI
"FB20_RA_AI"
BEGIN
   IN4 := 100.0;
   IN5 := 5.0;
   IN6 := 15.0;
   IN7 := 85.0;
   IN8 := 95.0;
END_DATA_BLOCK

DATA_BLOCK "DB153_HMI_FP1"   // DB153
{ S7_Optimized_Access := 'TRUE' }
VERSION : 0.1
// stored: InstanceOfName FB2_HMI_STATUS
"FB2_HMI_STATUS"
BEGIN
END_DATA_BLOCK

DATA_BLOCK "DB154_DATA_STATUS"   // DB154
{ S7_Optimized_Access := 'FALSE' }
VERSION : 0.1
   VAR
      STAT0_STATUS_FP_1 : Int;
      STAT1_STATUS_FP_2 : Int;
      STAT2_STATUS_ID_FAN : Int;
      STAT3_STATUS_LH_FD_FAN : Int;
      STAT4_STATUS_RH_FD_FAN : Int;
      STAT5_STATUS_LH_STOKER : Int;
      STAT6_STATUS_RH_STOKER : Int;
      STAT7_STATUS_LH_SWING_CHUTE : Int;
      STAT8_STATUS_RH_SWING_CHUTE : Int;
      STAT9_STATUS_ASH_VALVE_1 : Int;
      STAT10_STATUS_ASH_VALVE_2 : Int;
      STAT11_STATUS_ASH_CONVEYOR : Int;
      STAT12 : Int;
      STAT13 : Int;
      STAT14 : Int;
      STAT15 : Int;
      STAT16_STATUS_WETSCRUBBER : Int;
      STAT17 : Int;
      STAT18 : Int;
      STAT19 : Int;
      STAT20_STATUS_COAL_CONV_1 : Int;
      STAT21_STATUS_COAL_CONV_2 : Int;
   END_VAR
BEGIN
END_DATA_BLOCK

DATA_BLOCK "DB155_HMI_FP2"   // DB155
{ S7_Optimized_Access := 'TRUE' }
VERSION : 0.1
// stored: InstanceOfName FB2_HMI_STATUS
"FB2_HMI_STATUS"
BEGIN
END_DATA_BLOCK

DATA_BLOCK "DB156_HMI_ID"   // DB156
{ S7_Optimized_Access := 'TRUE' }
VERSION : 0.1
// stored: InstanceOfName FB2_HMI_STATUS
"FB2_HMI_STATUS"
BEGIN
END_DATA_BLOCK

DATA_BLOCK "DB157_HMI_LHFD"   // DB157
{ S7_Optimized_Access := 'TRUE' }
VERSION : 0.1
// stored: InstanceOfName FB2_HMI_STATUS
"FB2_HMI_STATUS"
BEGIN
END_DATA_BLOCK

DATA_BLOCK "DB158_HMI_RHFD"   // DB158
{ S7_Optimized_Access := 'TRUE' }
VERSION : 0.1
// stored: InstanceOfName FB2_HMI_STATUS
"FB2_HMI_STATUS"
BEGIN
END_DATA_BLOCK

DATA_BLOCK "DB159_HMI_LHSTOKER"   // DB159
{ S7_Optimized_Access := 'TRUE' }
VERSION : 0.1
// stored: InstanceOfName FB2_HMI_STATUS
"FB2_HMI_STATUS"
BEGIN
END_DATA_BLOCK

DATA_BLOCK "DB160_HMI_RHSTOKER"   // DB160
{ S7_Optimized_Access := 'TRUE' }
VERSION : 0.1
// stored: InstanceOfName FB2_HMI_STATUS
"FB2_HMI_STATUS"
BEGIN
END_DATA_BLOCK

DATA_BLOCK "DB161_HMI_LHSWING"   // DB161
{ S7_Optimized_Access := 'TRUE' }
VERSION : 0.1
// stored: InstanceOfName FB2_HMI_STATUS
"FB2_HMI_STATUS"
BEGIN
END_DATA_BLOCK

DATA_BLOCK "DB162_HMI_RHSWING"   // DB162
{ S7_Optimized_Access := 'TRUE' }
VERSION : 0.1
// stored: InstanceOfName FB2_HMI_STATUS
"FB2_HMI_STATUS"
BEGIN
END_DATA_BLOCK

DATA_BLOCK "DB163_HMI_ASHCONV"   // DB163
{ S7_Optimized_Access := 'TRUE' }
VERSION : 0.1
// stored: InstanceOfName FB2_HMI_STATUS
"FB2_HMI_STATUS"
BEGIN
END_DATA_BLOCK

DATA_BLOCK "DB164_HMI_ASH_V1"   // DB164
{ S7_Optimized_Access := 'TRUE' }
VERSION : 0.1
// stored: InstanceOfName FB2_HMI_STATUS
"FB2_HMI_STATUS"
BEGIN
END_DATA_BLOCK

DATA_BLOCK "DB165_HMI_ASH_V2"   // DB165
{ S7_Optimized_Access := 'TRUE' }
VERSION : 0.1
// stored: InstanceOfName FB2_HMI_STATUS
"FB2_HMI_STATUS"
BEGIN
END_DATA_BLOCK

DATA_BLOCK "DB170_HMI_WETSCRUB"   // DB170
{ S7_Optimized_Access := 'TRUE' }
VERSION : 0.1
// stored: InstanceOfName FB2_HMI_STATUS
"FB2_HMI_STATUS"
BEGIN
END_DATA_BLOCK

DATA_BLOCK "DB173_LHFD_SCALING"   // DB173
{ S7_Optimized_Access := 'TRUE' }
VERSION : 0.1
// stored: InstanceOfName FB20_RA_AI
"FB20_RA_AI"
BEGIN
   IN4 := 100.0;
   IN5 := 5.0;
   IN6 := 15.0;
   IN7 := 85.0;
   IN8 := 95.0;
END_DATA_BLOCK

DATA_BLOCK "DB176_RH_FD_SCALING"   // DB176
{ S7_Optimized_Access := 'TRUE' }
VERSION : 0.1
// stored: InstanceOfName FB20_RA_AI
"FB20_RA_AI"
BEGIN
   IN4 := 100.0;
   IN5 := 5.0;
   IN6 := 15.0;
   IN7 := 85.0;
   IN8 := 95.0;
END_DATA_BLOCK

DATA_BLOCK "DB183_LH_COAL_COUNTER"   // DB183
{ S7_Optimized_Access := 'TRUE' }
VERSION : 0.1
// stored: InstanceOfName FB3_COAL_COUNTER_FB
"FB3_COAL_COUNTER_FB"
BEGIN
END_DATA_BLOCK

DATA_BLOCK "DB184_RH_COAL_COUNTER"   // DB184
{ S7_Optimized_Access := 'TRUE' }
VERSION : 0.1
// stored: InstanceOfName FB3_COAL_COUNTER_FB
"FB3_COAL_COUNTER_FB"
BEGIN
END_DATA_BLOCK

DATA_BLOCK "DB185_AUTO_BLOWDOWN_DATA"   // DB185
{ S7_Optimized_Access := 'TRUE' }
VERSION : 0.1
// stored: InstanceOfName FB6_AUTO_BLOWDOWN
"FB6_AUTO_BLOWDOWN"
BEGIN
   IN1 := T#10s;
   IN2 := T#15s;
   IN0 := 480;
   IN3 := 3;
END_DATA_BLOCK

DATA_BLOCK "DB190_CONV1_HMI_STATUS"   // DB190
{ S7_Optimized_Access := 'TRUE' }
VERSION : 0.1
// stored: InstanceOfName FB2_HMI_STATUS
"FB2_HMI_STATUS"
BEGIN
END_DATA_BLOCK

DATA_BLOCK "DB191_CONV2_HMI_STATUS"   // DB191
{ S7_Optimized_Access := 'TRUE' }
VERSION : 0.1
// stored: InstanceOfName FB2_HMI_STATUS
"FB2_HMI_STATUS"
BEGIN
END_DATA_BLOCK

DATA_BLOCK "DB192_LH_STOKER_MM"   // DB192
{ S7_Optimized_Access := 'TRUE' }
VERSION : 0.1
// stored: InstanceOfName FB20_RA_AI
"FB20_RA_AI"
BEGIN
   IN4 := 136.0;
   IN5 := 5.0;
   IN6 := 15.0;
   IN7 := 85.0;
   IN8 := 95.0;
END_DATA_BLOCK

DATA_BLOCK "DB193_HAND SPEED REFF LH FD"   // DB193
{ S7_Optimized_Access := 'TRUE' }
VERSION : 0.1
// stored: InstanceOfName FB22_RA_AO_CUSTOM
"FB22_RA_AO_CUSTOM"
BEGIN
   IN4 := 50.0;
   IN5 := 5.0;
   IN6 := 15.0;
   IN7 := 85.0;
   IN8 := 95.0;
   IN3 := 46.0;
   IN13 := 11059.0;
   IN14 := 14376.0;
END_DATA_BLOCK

DATA_BLOCK "DB194_SPEED REFF RH FD FAN (HA"   // DB194
{ S7_Optimized_Access := 'TRUE' }
VERSION : 0.1
// stored: InstanceOfName FB22_RA_AO_CUSTOM
"FB22_RA_AO_CUSTOM"
BEGIN
   IN4 := 50.0;
   IN5 := 5.0;
   IN6 := 15.0;
   IN7 := 85.0;
   IN8 := 95.0;
   IN3 := 58.5;
   IN13 := 11059.0;
   IN14 := 13824.0;
END_DATA_BLOCK

DATA_BLOCK "DB196_SPEED REFF LH STOKER AUT"   // DB196
{ S7_Optimized_Access := 'TRUE' }
VERSION : 0.1
// stored: InstanceOfName FB22_RA_AO_CUSTOM
"FB22_RA_AO_CUSTOM"
BEGIN
   IN4 := 50.0;
   IN5 := 5.0;
   IN6 := 15.0;
   IN7 := 85.0;
   IN8 := 95.0;
   IN3 := 50.0;
   IN13 := 16588.0;
   IN14 := 22118.0;
END_DATA_BLOCK

DATA_BLOCK "DB197_SPEED REFF RH STOKER AUT"   // DB197
{ S7_Optimized_Access := 'TRUE' }
VERSION : 0.1
// stored: InstanceOfName FB22_RA_AO_CUSTOM
"FB22_RA_AO_CUSTOM"
BEGIN
   IN4 := 50.0;
   IN5 := 5.0;
   IN6 := 15.0;
   IN7 := 85.0;
   IN8 := 95.0;
   IN3 := 50.0;
   IN13 := 16588.0;
   IN14 := 22118.0;
END_DATA_BLOCK

DATA_BLOCK "DB198_LH_BUCKET_DB"   // DB198
{ S7_Optimized_Access := 'TRUE' }
VERSION : 0.1
// stored: InstanceOfName FB5_SINGLE_BUCKET
"FB5_SINGLE_BUCKET"
BEGIN
END_DATA_BLOCK

DATA_BLOCK "DB199_RH_BUCKET_DB"   // DB199
{ S7_Optimized_Access := 'TRUE' }
VERSION : 0.1
// stored: InstanceOfName FB5_SINGLE_BUCKET
"FB5_SINGLE_BUCKET"
BEGIN
   IN12 := T#7s;
END_DATA_BLOCK

DATA_BLOCK "DB201_STOKER_&_FD"   // DB201
{ S7_Optimized_Access := 'FALSE' }
VERSION : 0.1
   VAR
      STAT0_SP_STOKER : Real := 12.0;
      STAT1_GAIN_STOKER : Real := 10.0;
      STAT2_TI_STOKER : Real := 10.0;
      STAT3_TD_STOKER : Real := 10.0;
      STAT4_SUB_PID_OUT_FD_0 : Real := -4.5;
      STAT5_MAX_PID_OUT_FD : Real := 4.5;
      STAT6_Max_Perc_O2 : Real := 9.0;
      STAT7_MAX_PERC_CALC : Real := 0.09;
      STAT8_SP_FD_Fan : Real := 12.4;
      STAT9_GAIN_FD : Real := 1.0;
      STAT10_TI_FD : Real := 100.0;
      STAT11_TD_FD : Real := 0.1;
   END_VAR
BEGIN
END_DATA_BLOCK

// folder: System blocks/Program resources

DATA_BLOCK "T4"   // DB2
{ S7_Optimized_Access := 'TRUE' }
AUTHOR : Simatic
FAMILY : IEC
NAME : IEC_TMR
VERSION : 1.0
// stored: InstanceOfName IEC_TIMER
"IEC_TIMER"
BEGIN
END_DATA_BLOCK

DATA_BLOCK "T5"   // DB3
{ S7_Optimized_Access := 'TRUE' }
AUTHOR : Simatic
FAMILY : IEC
NAME : IEC_TMR
VERSION : 1.0
// stored: InstanceOfName IEC_TIMER
"IEC_TIMER"
BEGIN
END_DATA_BLOCK

DATA_BLOCK "T18"   // DB5
{ S7_Optimized_Access := 'TRUE' }
AUTHOR : Simatic
FAMILY : IEC
NAME : IEC_TMR
VERSION : 1.0
// stored: InstanceOfName IEC_TIMER
"IEC_TIMER"
BEGIN
END_DATA_BLOCK

DATA_BLOCK "T19"   // DB6
{ S7_Optimized_Access := 'TRUE' }
AUTHOR : Simatic
FAMILY : IEC
NAME : IEC_TMR
VERSION : 1.0
// stored: InstanceOfName IEC_TIMER
"IEC_TIMER"
BEGIN
END_DATA_BLOCK

DATA_BLOCK "T20"   // DB7
{ S7_Optimized_Access := 'TRUE' }
AUTHOR : Simatic
FAMILY : IEC
NAME : IEC_TMR
VERSION : 1.0
// stored: InstanceOfName IEC_TIMER
"IEC_TIMER"
BEGIN
END_DATA_BLOCK

DATA_BLOCK "T21"   // DB8
{ S7_Optimized_Access := 'TRUE' }
AUTHOR : Simatic
FAMILY : IEC
NAME : IEC_TMR
VERSION : 1.0
// stored: InstanceOfName IEC_TIMER
"IEC_TIMER"
BEGIN
END_DATA_BLOCK

DATA_BLOCK "T2"   // DB10
{ S7_Optimized_Access := 'TRUE' }
AUTHOR : Simatic
FAMILY : IEC
NAME : IEC_TMR
VERSION : 1.0
// stored: InstanceOfName IEC_TIMER
"IEC_TIMER"
BEGIN
END_DATA_BLOCK

DATA_BLOCK "T3"   // DB11
{ S7_Optimized_Access := 'TRUE' }
AUTHOR : Simatic
FAMILY : IEC
NAME : IEC_TMR
VERSION : 1.0
// stored: InstanceOfName IEC_TIMER
"IEC_TIMER"
BEGIN
END_DATA_BLOCK

DATA_BLOCK "T6"   // DB12
{ S7_Optimized_Access := 'TRUE' }
AUTHOR : Simatic
FAMILY : IEC
NAME : IEC_TMR
VERSION : 1.0
// stored: InstanceOfName IEC_TIMER
"IEC_TIMER"
BEGIN
END_DATA_BLOCK

DATA_BLOCK "T7"   // DB13
{ S7_Optimized_Access := 'TRUE' }
AUTHOR : Simatic
FAMILY : IEC
NAME : IEC_TMR
VERSION : 1.0
// stored: InstanceOfName IEC_TIMER
"IEC_TIMER"
BEGIN
END_DATA_BLOCK

DATA_BLOCK "T1"   // DB14
{ S7_Optimized_Access := 'TRUE' }
AUTHOR : Simatic
FAMILY : IEC
NAME : IEC_TMR
VERSION : 1.0
// stored: InstanceOfName IEC_TIMER
"IEC_TIMER"
BEGIN
END_DATA_BLOCK

DATA_BLOCK "T14"   // DB15
{ S7_Optimized_Access := 'TRUE' }
AUTHOR : Simatic
FAMILY : IEC
NAME : IEC_TMR
VERSION : 1.0
// stored: InstanceOfName IEC_TIMER
"IEC_TIMER"
BEGIN
END_DATA_BLOCK

DATA_BLOCK "T15"   // DB16
{ S7_Optimized_Access := 'TRUE' }
AUTHOR : Simatic
FAMILY : IEC
NAME : IEC_TMR
VERSION : 1.0
// stored: InstanceOfName IEC_TIMER
"IEC_TIMER"
BEGIN
END_DATA_BLOCK

DATA_BLOCK "T16"   // DB17
{ S7_Optimized_Access := 'TRUE' }
AUTHOR : Simatic
FAMILY : IEC
NAME : IEC_TMR
VERSION : 1.0
// stored: InstanceOfName IEC_TIMER
"IEC_TIMER"
BEGIN
END_DATA_BLOCK

DATA_BLOCK "T8"   // DB18
{ S7_Optimized_Access := 'TRUE' }
AUTHOR : Simatic
FAMILY : IEC
NAME : IEC_TMR
VERSION : 1.0
// stored: InstanceOfName IEC_TIMER
"IEC_TIMER"
BEGIN
END_DATA_BLOCK

DATA_BLOCK "T9"   // DB19
{ S7_Optimized_Access := 'TRUE' }
AUTHOR : Simatic
FAMILY : IEC
NAME : IEC_TMR
VERSION : 1.0
// stored: InstanceOfName IEC_TIMER
"IEC_TIMER"
BEGIN
END_DATA_BLOCK

DATA_BLOCK "T23"   // DB20
{ S7_Optimized_Access := 'TRUE' }
AUTHOR : Simatic
FAMILY : IEC
NAME : IEC_TMR
VERSION : 1.0
// stored: InstanceOfName IEC_TIMER
"IEC_TIMER"
BEGIN
END_DATA_BLOCK

// folder: (top level)

FUNCTION_BLOCK "FB1_HZ_TO_PERCENT"   // FB1, LAD
{ S7_Optimized_Access := 'TRUE' }
VERSION : 0.1
   VAR_INPUT
      IN0 : Real;
      IN1 : Real;
   END_VAR
   VAR_OUTPUT
      Out2 : Real;
   END_VAR
   VAR
      STAT3 : Real;
   END_VAR
BEGIN

REGION Network 1
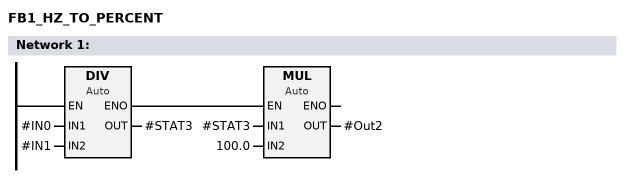
   RUNG wire#powerrail
      Div(in1 := #IN0, in2 := #IN1, out => #STAT3)
      Mul(in1 := #STAT3, in2 := 100.0, out => #Out2)
   END_RUNG
   // the same network as SCL:
   #STAT3 := #IN0 / #IN1;
   #Out2 := #STAT3 * 100.0;
END_REGION
END_FUNCTION_BLOCK

FUNCTION_BLOCK "FB2_HMI_STATUS"   // FB2, LAD
{ S7_Optimized_Access := 'TRUE' }
VERSION : 0.1
   VAR_INPUT
      IN0 : Bool;
      IN1 : Bool;
      IN2 : Bool;
      IN3 : Bool;
   END_VAR
   VAR_OUTPUT
      Out4 : Int;
   END_VAR
BEGIN

REGION Network 1
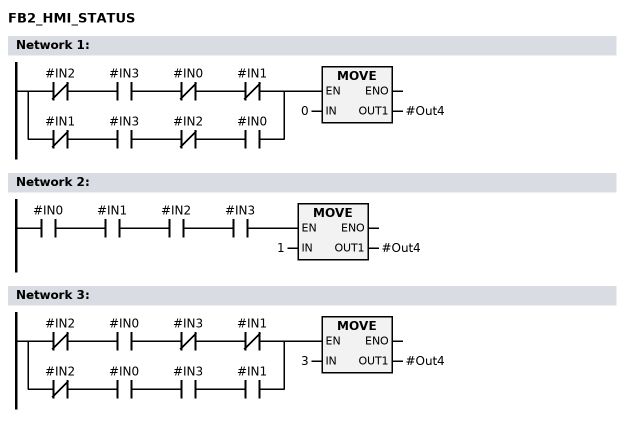
   RUNG wire#powerrail
      I_Contact( #IN2 )
      Contact( #IN3 )
      I_Contact( #IN0 )
      I_Contact( #IN1 )
      wire#w1
      Move(in := 0, out1 => #Out4)
   END_RUNG
   RUNG wire#powerrail
      I_Contact( #IN1 )
      Contact( #IN3 )
      I_Contact( #IN2 )
      Contact( #IN0 )
   END_RUNG wire#w1
   // the same network as SCL:
   IF (NOT #IN2 AND #IN3 AND NOT #IN0 AND NOT #IN1) OR (NOT #IN1 AND #IN3 AND NOT #IN2 AND #IN0) THEN
       #Out4 := 0;
   END_IF;
END_REGION

REGION Network 2
   RUNG wire#powerrail
      Contact( #IN0 )
      Contact( #IN1 )
      Contact( #IN2 )
      Contact( #IN3 )
      Move(in := 1, out1 => #Out4)
   END_RUNG
   // the same network as SCL:
   IF #IN0 AND #IN1 AND #IN2 AND #IN3 THEN #Out4 := 1; END_IF;
END_REGION

REGION Network 3
   RUNG wire#powerrail
      I_Contact( #IN2 )
      Contact( #IN0 )
      I_Contact( #IN3 )
      I_Contact( #IN1 )
      wire#w1
      Move(in := 3, out1 => #Out4)
   END_RUNG
   RUNG wire#powerrail
      I_Contact( #IN2 )
      Contact( #IN0 )
      Contact( #IN3 )
      Contact( #IN1 )
   END_RUNG wire#w1
   // the same network as SCL:
   IF (NOT #IN2 AND #IN0 AND NOT #IN3 AND NOT #IN1) OR (NOT #IN2 AND #IN0 AND #IN3 AND #IN1) THEN
       #Out4 := 3;
   END_IF;
END_REGION
END_FUNCTION_BLOCK

FUNCTION_BLOCK "FB3_COAL_COUNTER_FB"   // FB3, LAD
TITLE = coal counter fb
{ S7_Optimized_Access := 'TRUE' }
VERSION : 0.1
// counting coal use
   VAR_INPUT
      IN0 : Real;
      IN1 : Real;
      IN2 : Bool;
   END_VAR
   VAR_OUTPUT
      Out4 : Real;
   END_VAR
   VAR
      STAT6 : Real;
      STAT7 : Real;
      STAT8 : Real;
      STAT9 : DInt;
      STAT10 : DInt;
      STAT16 : Bool;
      STAT15 : Bool;
      STAT13 : Real;
      IN3 : TON_TIME;
   END_VAR
   VAR_TEMP   // added for the SCL form of the ladder/FBD networks
      _w1 : Bool;
      _w2 : Bool;
   END_VAR
BEGIN

REGION Network 1
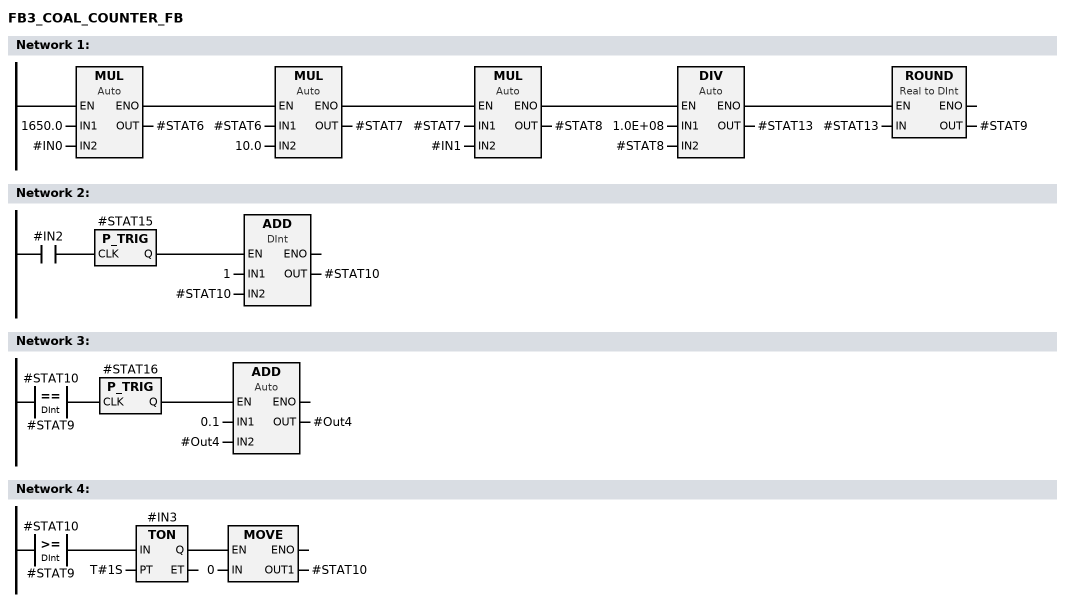
   RUNG wire#powerrail
      Mul(in1 := 1650.0, in2 := #IN0, out => #STAT6)
      Mul(in1 := #STAT6, in2 := 10.0, out => #STAT7)
      Mul(in1 := #STAT7, in2 := #IN1, out => #STAT8)
      Div(in1 := 1.0E+08, in2 := #STAT8, out => #STAT13)
      { S7_Templates := "[SrcType := Real, DestType := DInt]" } Round(in := #STAT13, out => #STAT9)
   END_RUNG
   // the same network as SCL:
   #STAT6 := 1650.0 * #IN0;
   #STAT7 := #STAT6 * 10.0;
   #STAT8 := #STAT7 * #IN1;
   #STAT13 := 1.0E+08 / #STAT8;
   #STAT9 := ROUND(#STAT13);
END_REGION

REGION Network 2
   RUNG wire#powerrail
      Contact( #IN2 )
      P_Trig( #STAT15 )
      { S7_Templates := "SrcType := DInt" } Add(in1 := 1, in2 := #STAT10, out => #STAT10)
   END_RUNG
   // the same network as SCL:
   #_w1 := #IN2 AND NOT #STAT15;   // rising edge
   #STAT15 := #IN2;
   IF #_w1 THEN #STAT10 := 1 + #STAT10; END_IF;
END_REGION

REGION Network 3
   RUNG wire#powerrail
      { S7_Templates := "SrcType := DInt" } EQ_Contact(in1 := #STAT10, in2 := #STAT9)
      P_Trig( #STAT16 )
      Add(in1 := 0.1, in2 := #Out4, out => #Out4)
   END_RUNG
   // the same network as SCL:
   #_w1 := #STAT10 = #STAT9;
   #_w2 := #_w1 AND NOT #STAT16;   // rising edge
   #STAT16 := #_w1;
   IF #_w2 THEN #Out4 := 0.1 + #Out4; END_IF;
END_REGION

REGION Network 4
   #IN3(IN := #STAT10 >= #STAT9, PT := T#1S);   // TON
   IF #IN3.Q THEN #STAT10 := 0; END_IF;
END_REGION
END_FUNCTION_BLOCK

FUNCTION_BLOCK "FB5_SINGLE_BUCKET"   // FB5, LAD
{ S7_Optimized_Access := 'TRUE' }
VERSION : 0.1
   VAR_INPUT
      IN0 : Bool;
      IN1 : Bool;
      IN2 : Bool;
      IN3 : Bool;
      IN4 : Bool;
      IN5 : Bool;
      IN6 : Bool;
      IN7 : Bool;
      IN8 : Bool;
      IN9 : Bool;
      IN10 : Bool;
      IN12 : Time;
   END_VAR
   VAR_IN_OUT
      IO13 : Bool;
      IO14 : Bool;
   END_VAR
   VAR
      STAT15 : Bool;
      IN11 : TON_TIME;
   END_VAR
   VAR_TEMP   // added for the SCL form of the ladder/FBD networks
      _w1 : Bool;
   END_VAR
BEGIN

REGION Network 1
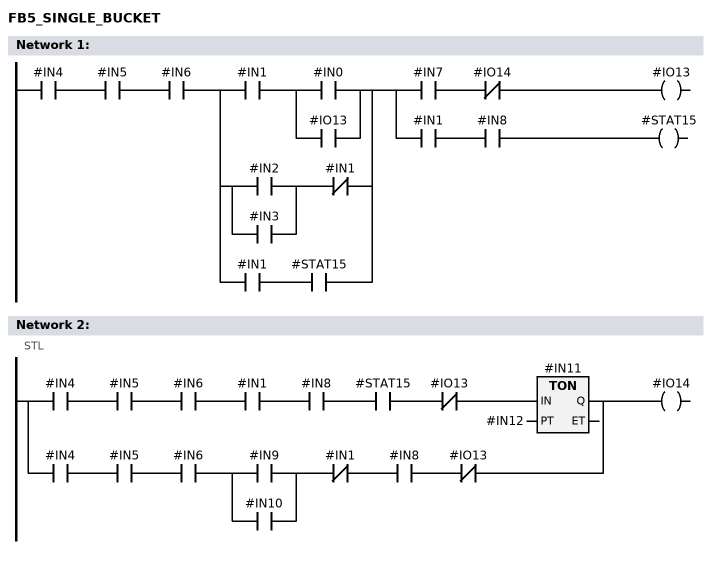
   RUNG wire#powerrail
      Contact( #IN4 )
      Contact( #IN5 )
      Contact( #IN6 )
      wire#w1
      Contact( #IN1 )
      wire#w2
      Contact( #IN0 )
      wire#w3
      Contact( #IN7 )
      I_Contact( #IO14 )
      Coil( #IO13 )
   END_RUNG
   RUNG wire#w2
      Contact( #IO13 )
   END_RUNG wire#w3
   RUNG wire#w1
      Contact( #IN2 )
      wire#w4
      I_Contact( #IN1 )
   END_RUNG wire#w3
   RUNG wire#w1
      Contact( #IN3 )
   END_RUNG wire#w4
   RUNG wire#w1
      Contact( #IN1 )
      Contact( #STAT15 )
   END_RUNG wire#w3
   RUNG wire#w3
      Contact( #IN1 )
      Contact( #IN8 )
      Coil( #STAT15 )
   END_RUNG
   // the same network as SCL:
   #_w1 := #IN4 AND #IN5 AND #IN6 AND ((#IN1 AND (#IN0 OR #IO13)) OR ((#IN2 OR #IN3) AND NOT #IN1) OR (#IN1 AND #STAT15));
   #IO13 := #_w1 AND #IN7 AND NOT #IO14;
   #STAT15 := #_w1 AND #IN1 AND #IN8;
END_REGION

REGION Network 2
   // STL
   #IN11(IN := #IN4 AND #IN5 AND #IN6 AND #IN1 AND #IN8 AND #STAT15 AND NOT #IO13, PT := #IN12);   // TON
   #IO14 := #IN11.Q OR (#IN4 AND #IN5 AND #IN6 AND (#IN9 OR #IN10) AND NOT #IN1 AND #IN8 AND NOT #IO13);
END_REGION
END_FUNCTION_BLOCK

FUNCTION_BLOCK "FB6_AUTO_BLOWDOWN"   // FB6, LAD
{ S7_Optimized_Access := 'TRUE' }
VERSION : 0.1
   VAR_INPUT
      IN0 : Int;
      IN1 : Time;
      IN2 : Time;
      IN3 : Int;
   END_VAR
   VAR_OUTPUT
      Out4 : Bool;
   END_VAR
   VAR
      STAT5 : Int;
      STAT6 : Int;
      STAT7 : Bool;
      STAT8 : Int;
      STAT9 : Bool;
      STAT10 : Bool;
   END_VAR
   VAR_TEMP   // added for the SCL form of the ladder/FBD networks
      _w1 : Bool;
   END_VAR
BEGIN

REGION Network 1: Counting Second
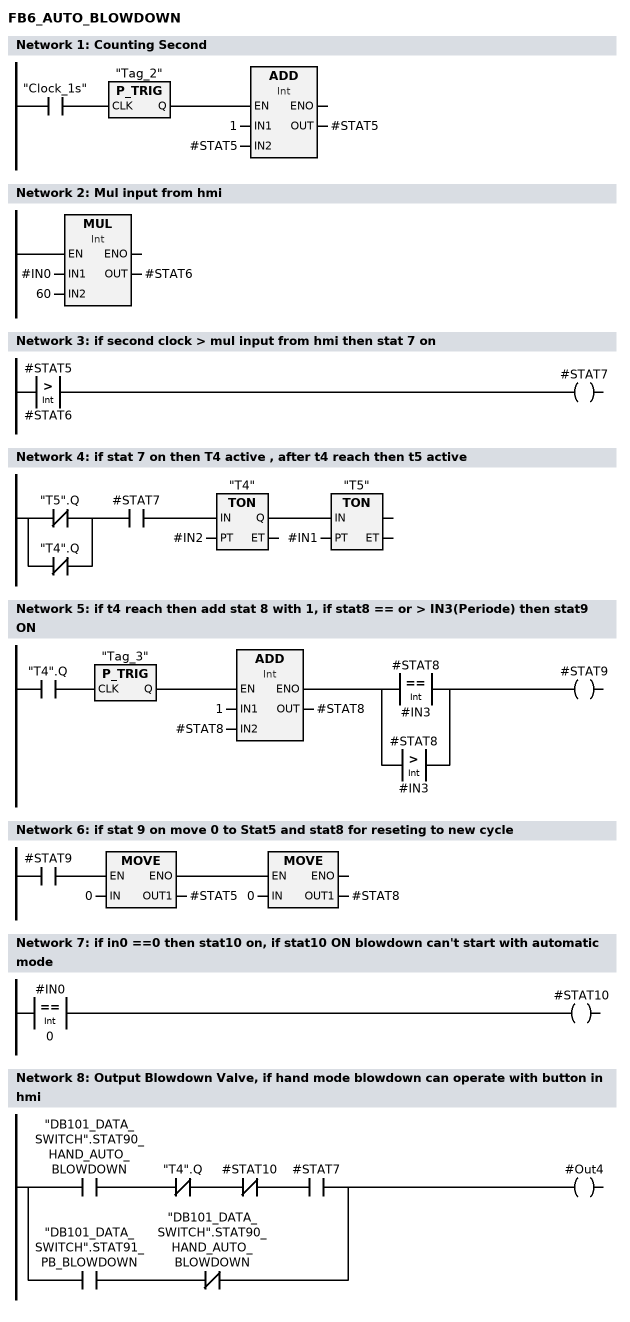
   RUNG wire#powerrail
      Contact( "Clock_1s" )
      P_Trig( "Tag_2" )
      { S7_Templates := "SrcType := Int" } Add(in1 := 1, in2 := #STAT5, out => #STAT5)
   END_RUNG
   // the same network as SCL:
   #_w1 := "Clock_1s" AND NOT "Tag_2";   // rising edge
   "Tag_2" := "Clock_1s";
   IF #_w1 THEN #STAT5 := 1 + #STAT5; END_IF;
END_REGION

REGION Network 2: Mul input from hmi
   RUNG wire#powerrail
      { S7_Templates := "SrcType := Int" } Mul(in1 := #IN0, in2 := 60, out => #STAT6)
   END_RUNG
   // the same network as SCL:
   #STAT6 := #IN0 * 60;
END_REGION

REGION Network 3: if second clock > mul input from hmi then stat 7 on
   RUNG wire#powerrail
      { S7_Templates := "SrcType := Int" } GT_Contact(in1 := #STAT5, in2 := #STAT6)
      Coil( #STAT7 )
   END_RUNG
   // the same network as SCL:
   #STAT7 := #STAT5 > #STAT6;
END_REGION

REGION Network 4: if stat 7 on then T4 active , after t4 reach then t5 active
   "T4".TON(IN := (NOT "T5".Q OR NOT "T4".Q) AND #STAT7, PT := #IN2);
   "T5".TON(IN := "T4".Q, PT := #IN1);
END_REGION

REGION Network 5: if t4 reach then add stat 8 with 1, if stat8 == or > IN3(Periode) then stat9 ON
   RUNG wire#powerrail
      Contact( "T4".Q )
      P_Trig( "Tag_3" )
      { S7_Templates := "SrcType := Int" } Add(in1 := 1, in2 := #STAT8, out => #STAT8)
      wire#w1
      { S7_Templates := "SrcType := Int" } EQ_Contact(in1 := #STAT8, in2 := #IN3)
      wire#w2
      Coil( #STAT9 )
   END_RUNG
   RUNG wire#w1
      { S7_Templates := "SrcType := Int" } GT_Contact(in1 := #STAT8, in2 := #IN3)
   END_RUNG wire#w2
   // the same network as SCL:
   #_w1 := "T4".Q AND NOT "Tag_3";   // rising edge
   "Tag_3" := "T4".Q;
   IF #_w1 THEN #STAT8 := 1 + #STAT8; END_IF;
   #STAT9 := #_w1 AND ((#STAT8 = #IN3) OR (#STAT8 > #IN3));
END_REGION

REGION Network 6: if stat 9 on move 0 to Stat5 and stat8 for reseting to new cycle
   RUNG wire#powerrail
      Contact( #STAT9 )
      Move(in := 0, out1 => #STAT5)
      Move(in := 0, out1 => #STAT8)
   END_RUNG
   // the same network as SCL:
   IF #STAT9 THEN
       #STAT5 := 0;
       #STAT8 := 0;
   END_IF;
END_REGION

REGION Network 7: if in0 ==0 then stat10 on, if stat10 ON blowdown can't start with automatic mode
   RUNG wire#powerrail
      { S7_Templates := "SrcType := Int" } EQ_Contact(in1 := #IN0, in2 := 0)
      Coil( #STAT10 )
   END_RUNG
   // the same network as SCL:
   #STAT10 := #IN0 = 0;
END_REGION

REGION Network 8: Output Blowdown Valve, if hand mode blowdown can operate with button in hmi
   RUNG wire#powerrail
      Contact( "DB101_DATA_SWITCH".STAT90_HAND_AUTO_BLOWDOWN )
      I_Contact( "T4".Q )
      I_Contact( #STAT10 )
      Contact( #STAT7 )
      wire#w1
      Coil( #Out4 )
   END_RUNG
   RUNG wire#powerrail
      Contact( "DB101_DATA_SWITCH".STAT91_PB_BLOWDOWN )
      I_Contact( "DB101_DATA_SWITCH".STAT90_HAND_AUTO_BLOWDOWN )
   END_RUNG wire#w1
   // the same network as SCL:
   #Out4 := ("DB101_DATA_SWITCH".STAT90_HAND_AUTO_BLOWDOWN AND NOT "T4".Q AND NOT #STAT10 AND #STAT7) OR ("DB101_DATA_SWITCH".STAT91_PB_BLOWDOWN AND NOT "DB101_DATA_SWITCH".STAT90_HAND_AUTO_BLOWDOWN);
END_REGION
END_FUNCTION_BLOCK

FUNCTION_BLOCK "FB20_RA_AI"   // FB20, LAD
{ S7_Optimized_Access := 'TRUE' }
VERSION : 0.1
   VAR_INPUT
      IN0 : Bool;
      IN1 : Bool;
      IN2 : Int;
      IN3 : Real;
      IN4 : Real;
      IN5 : Real;
      IN6 : Real;
      IN7 : Real;
      IN8 : Real;
      IN9 : Bool;
      IN10 : Bool;
      IN11 : Bool;
      IN12 : Bool;
   END_VAR
   VAR_OUTPUT
      Out13 : Real;
      Out14 : Bool;
      Out15 : Bool;
      Out16 : Bool;
      Out17 : Bool;
      Out18 : Bool;
   END_VAR
   VAR_IN_OUT
      IO19 : Real;
   END_VAR
   VAR_TEMP
      Temp20 : Word;
      INN2 : Int;
   END_VAR
BEGIN

REGION Network 1
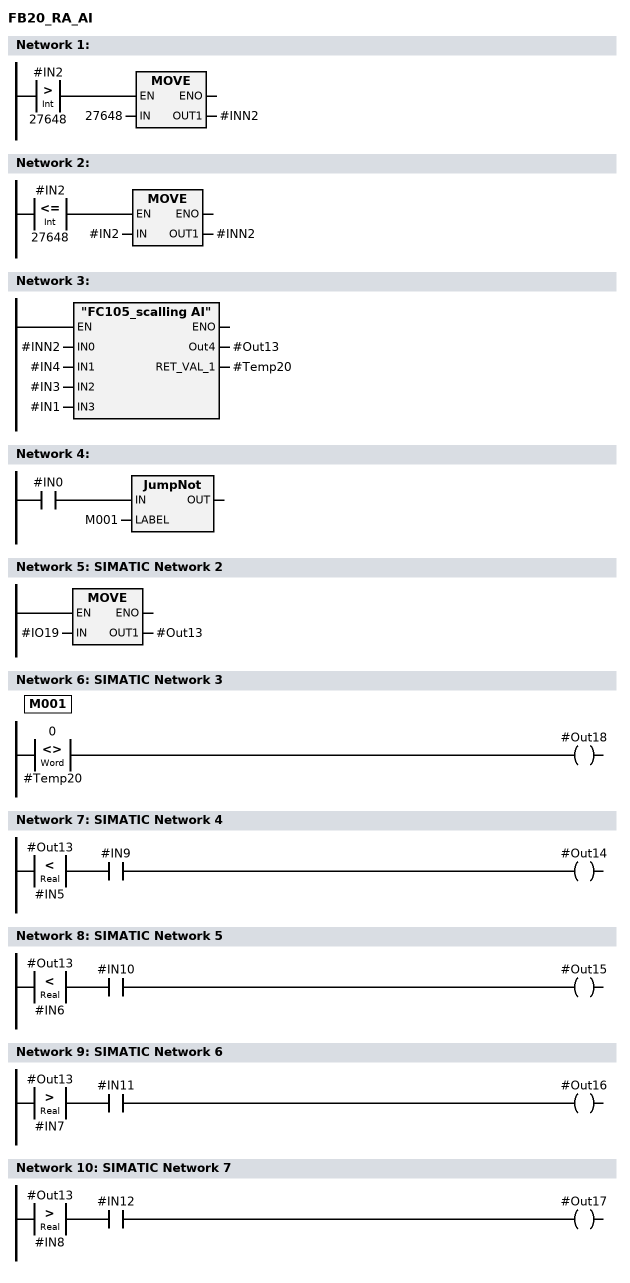
   RUNG wire#powerrail
      { S7_Templates := "SrcType := Int" } GT_Contact(in1 := #IN2, in2 := 27648)
      Move(in := 27648, out1 => #INN2)
   END_RUNG
   // the same network as SCL:
   IF #IN2 > 27648 THEN #INN2 := 27648; END_IF;
END_REGION

REGION Network 2
   RUNG wire#powerrail
      { S7_Templates := "SrcType := Int" } LE_Contact(in1 := #IN2, in2 := 27648)
      Move(in := #IN2, out1 => #INN2)
   END_RUNG
   // the same network as SCL:
   IF #IN2 <= 27648 THEN #INN2 := #IN2; END_IF;
END_REGION

REGION Network 3
   RUNG wire#powerrail
      "FC105_scalling AI"(IN0 := #INN2, IN1 := #IN4, IN2 := #IN3, IN3 := #IN1, Out4 => #Out13, RET_VAL_1 => #Temp20)
   END_RUNG
   // the same network as SCL:
   "FC105_scalling AI"(IN0 := #INN2,
                       IN1 := #IN4,
                       IN2 := #IN3,
                       IN3 := #IN1,
                       Out4 => #Out13,
                       RET_VAL_1 => #Temp20);
END_REGION

REGION Network 4
   // no SCL statement known for JumpNot: written as a call
   JumpNot(in := #IN0, label := M001);
END_REGION

REGION Network 5: SIMATIC Network 2
   RUNG wire#powerrail
      Move(in := #IO19, out1 => #Out13)
   END_RUNG
   // the same network as SCL:
   #Out13 := #IO19;
END_REGION

REGION Network 6: SIMATIC Network 3
   Label( M001 )
   RUNG wire#powerrail
      { S7_Templates := "SrcType := Word" } NE_Contact(in1 := 0, in2 := #Temp20)
      Coil( #Out18 )
   END_RUNG
   // the same network as SCL:
   M001:
   #Out18 := 0 <> #Temp20;
END_REGION

REGION Network 7: SIMATIC Network 4
   RUNG wire#powerrail
      { S7_Templates := "SrcType := Real" } LT_Contact(in1 := #Out13, in2 := #IN5)
      Contact( #IN9 )
      Coil( #Out14 )
   END_RUNG
   // the same network as SCL:
   #Out14 := (#Out13 < #IN5) AND #IN9;
END_REGION

REGION Network 8: SIMATIC Network 5
   RUNG wire#powerrail
      { S7_Templates := "SrcType := Real" } LT_Contact(in1 := #Out13, in2 := #IN6)
      Contact( #IN10 )
      Coil( #Out15 )
   END_RUNG
   // the same network as SCL:
   #Out15 := (#Out13 < #IN6) AND #IN10;
END_REGION

REGION Network 9: SIMATIC Network 6
   RUNG wire#powerrail
      { S7_Templates := "SrcType := Real" } GT_Contact(in1 := #Out13, in2 := #IN7)
      Contact( #IN11 )
      Coil( #Out16 )
   END_RUNG
   // the same network as SCL:
   #Out16 := (#Out13 > #IN7) AND #IN11;
END_REGION

REGION Network 10: SIMATIC Network 7
   RUNG wire#powerrail
      { S7_Templates := "SrcType := Real" } GT_Contact(in1 := #Out13, in2 := #IN8)
      Contact( #IN12 )
      Coil( #Out17 )
   END_RUNG
   // the same network as SCL:
   #Out17 := (#Out13 > #IN8) AND #IN12;
END_REGION
END_FUNCTION_BLOCK

FUNCTION_BLOCK "FB21_RA_AO"   // FB21, LAD
{ S7_Optimized_Access := 'TRUE' }
VERSION : 0.1
   VAR_INPUT
      IN0 : Bool;
      IN1 : Bool;
      IN3 : Real;
      IN4 : Real;
      IN5 : Real;
      IN6 : Real;
      IN7 : Real;
      IN8 : Real;
      IN9 : Bool;
      IN10 : Bool;
      IN11 : Bool;
      IN12 : Bool;
   END_VAR
   VAR_OUTPUT
      Out13 : Int;
      Out14 : Bool;
      Out15 : Bool;
      Out16 : Bool;
      Out17 : Bool;
      Out18 : Bool;
   END_VAR
   VAR_IN_OUT
      IN2 : Real;
      IO19 : Real;
   END_VAR
   VAR_TEMP
      Temp20 : Word;
   END_VAR
BEGIN

REGION Network 1: SIMATIC Network 1
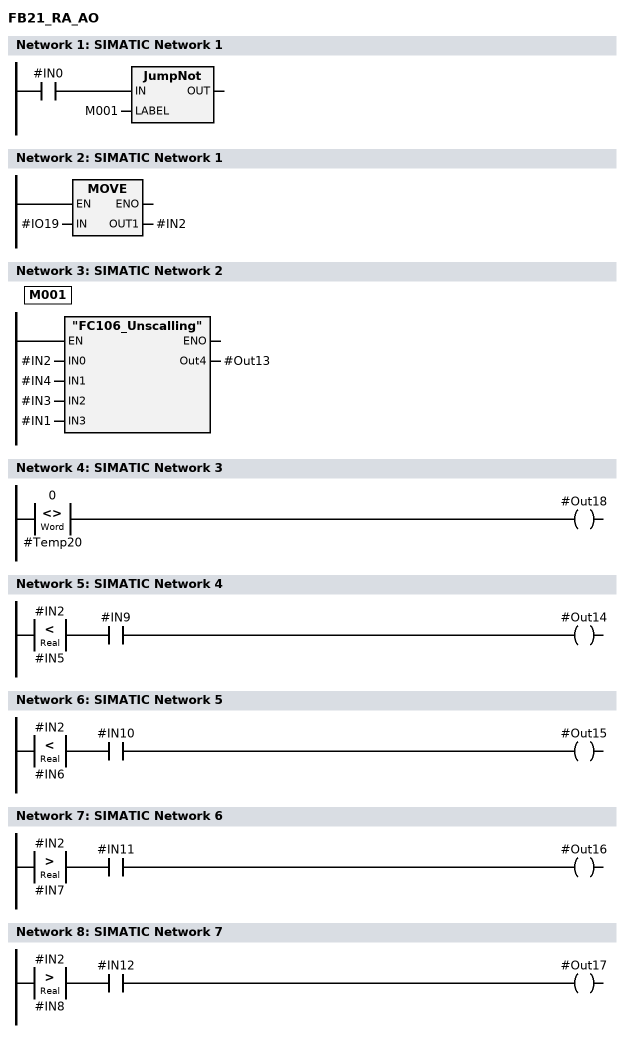
   // no SCL statement known for JumpNot: written as a call
   JumpNot(in := #IN0, label := M001);
END_REGION

REGION Network 2: SIMATIC Network 1
   RUNG wire#powerrail
      Move(in := #IO19, out1 => #IN2)
   END_RUNG
   // the same network as SCL:
   #IN2 := #IO19;
END_REGION

REGION Network 3: SIMATIC Network 2
   Label( M001 )
   RUNG wire#powerrail
      "FC106_Unscalling"(IN0 := #IN2, IN1 := #IN4, IN2 := #IN3, IN3 := #IN1, Out4 => #Out13)
   END_RUNG
   // the same network as SCL:
   M001:
   "FC106_Unscalling"(IN0 := #IN2, IN1 := #IN4, IN2 := #IN3, IN3 := #IN1, Out4 => #Out13);
END_REGION

REGION Network 4: SIMATIC Network 3
   RUNG wire#powerrail
      { S7_Templates := "SrcType := Word" } NE_Contact(in1 := 0, in2 := #Temp20)
      Coil( #Out18 )
   END_RUNG
   // the same network as SCL:
   #Out18 := 0 <> #Temp20;
END_REGION

REGION Network 5: SIMATIC Network 4
   RUNG wire#powerrail
      { S7_Templates := "SrcType := Real" } LT_Contact(in1 := #IN2, in2 := #IN5)
      Contact( #IN9 )
      Coil( #Out14 )
   END_RUNG
   // the same network as SCL:
   #Out14 := (#IN2 < #IN5) AND #IN9;
END_REGION

REGION Network 6: SIMATIC Network 5
   RUNG wire#powerrail
      { S7_Templates := "SrcType := Real" } LT_Contact(in1 := #IN2, in2 := #IN6)
      Contact( #IN10 )
      Coil( #Out15 )
   END_RUNG
   // the same network as SCL:
   #Out15 := (#IN2 < #IN6) AND #IN10;
END_REGION

REGION Network 7: SIMATIC Network 6
   RUNG wire#powerrail
      { S7_Templates := "SrcType := Real" } GT_Contact(in1 := #IN2, in2 := #IN7)
      Contact( #IN11 )
      Coil( #Out16 )
   END_RUNG
   // the same network as SCL:
   #Out16 := (#IN2 > #IN7) AND #IN11;
END_REGION

REGION Network 8: SIMATIC Network 7
   RUNG wire#powerrail
      { S7_Templates := "SrcType := Real" } GT_Contact(in1 := #IN2, in2 := #IN8)
      Contact( #IN12 )
      Coil( #Out17 )
   END_RUNG
   // the same network as SCL:
   #Out17 := (#IN2 > #IN8) AND #IN12;
END_REGION
END_FUNCTION_BLOCK

FUNCTION_BLOCK "FB22_RA_AO_CUSTOM"   // FB22, LAD
{ S7_Optimized_Access := 'TRUE' }
VERSION : 0.1
   VAR_INPUT
      IN0 : Bool;
      IN1 : Bool;
      IN3 : Real;
      IN4 : Real;
      IN5 : Real;
      IN6 : Real;
      IN7 : Real;
      IN8 : Real;
      IN9 : Bool;
      IN10 : Bool;
      IN11 : Bool;
      IN12 : Bool;
      IN13 : Real;
      IN14 : Real;
   END_VAR
   VAR_OUTPUT
      Out15 : Int;
      Out16 : Bool;
      Out17 : Bool;
      Out18 : Bool;
      Out19 : Bool;
      Out20 : Bool;
   END_VAR
   VAR_IN_OUT
      IO21 : Real;
      IN2 : Real;
   END_VAR
   VAR_TEMP
      Temp22 : Word;
   END_VAR
BEGIN

REGION Network 1
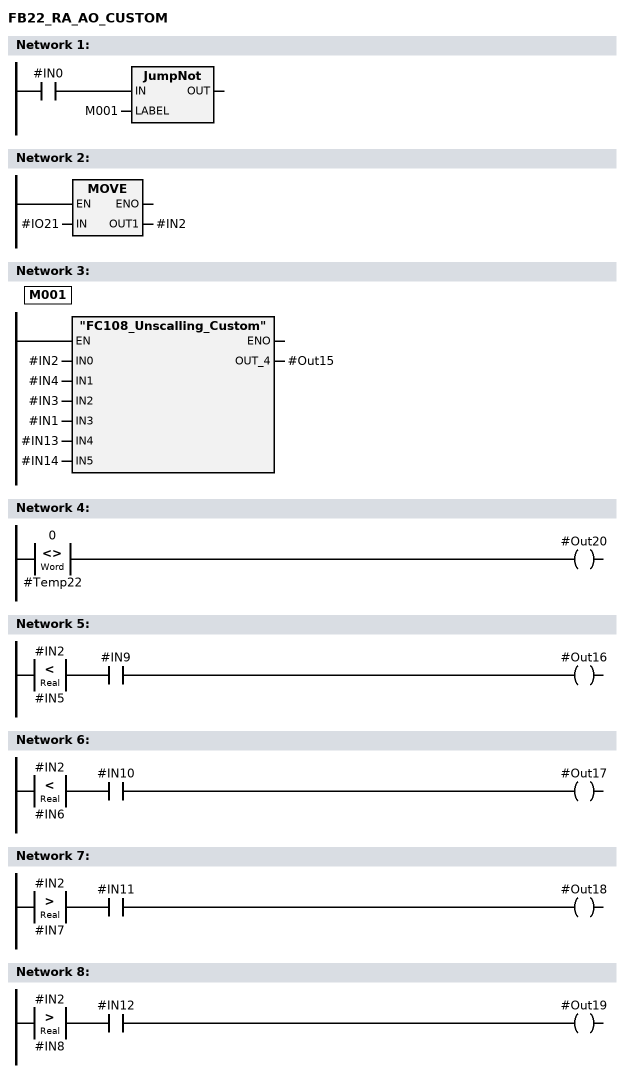
   // no SCL statement known for JumpNot: written as a call
   JumpNot(in := #IN0, label := M001);
END_REGION

REGION Network 2
   RUNG wire#powerrail
      Move(in := #IO21, out1 => #IN2)
   END_RUNG
   // the same network as SCL:
   #IN2 := #IO21;
END_REGION

REGION Network 3
   Label( M001 )
   RUNG wire#powerrail
      "FC108_Unscalling_Custom"(IN0 := #IN2, IN1 := #IN4, IN2 := #IN3, IN3 := #IN1, IN4 := #IN13, IN5 := #IN14, OUT_4 => #Out15)
   END_RUNG
   // the same network as SCL:
   M001:
   "FC108_Unscalling_Custom"(IN0 := #IN2,
                           IN1 := #IN4,
                           IN2 := #IN3,
                           IN3 := #IN1,
                           IN4 := #IN13,
                           IN5 := #IN14,
                           OUT_4 => #Out15);
END_REGION

REGION Network 4
   RUNG wire#powerrail
      { S7_Templates := "SrcType := Word" } NE_Contact(in1 := 0, in2 := #Temp22)
      Coil( #Out20 )
   END_RUNG
   // the same network as SCL:
   #Out20 := 0 <> #Temp22;
END_REGION

REGION Network 5
   RUNG wire#powerrail
      { S7_Templates := "SrcType := Real" } LT_Contact(in1 := #IN2, in2 := #IN5)
      Contact( #IN9 )
      Coil( #Out16 )
   END_RUNG
   // the same network as SCL:
   #Out16 := (#IN2 < #IN5) AND #IN9;
END_REGION

REGION Network 6
   RUNG wire#powerrail
      { S7_Templates := "SrcType := Real" } LT_Contact(in1 := #IN2, in2 := #IN6)
      Contact( #IN10 )
      Coil( #Out17 )
   END_RUNG
   // the same network as SCL:
   #Out17 := (#IN2 < #IN6) AND #IN10;
END_REGION

REGION Network 7
   RUNG wire#powerrail
      { S7_Templates := "SrcType := Real" } GT_Contact(in1 := #IN2, in2 := #IN7)
      Contact( #IN11 )
      Coil( #Out18 )
   END_RUNG
   // the same network as SCL:
   #Out18 := (#IN2 > #IN7) AND #IN11;
END_REGION

REGION Network 8
   RUNG wire#powerrail
      { S7_Templates := "SrcType := Real" } GT_Contact(in1 := #IN2, in2 := #IN8)
      Contact( #IN12 )
      Coil( #Out19 )
   END_RUNG
   // the same network as SCL:
   #Out19 := (#IN2 > #IN8) AND #IN12;
END_REGION
END_FUNCTION_BLOCK

FUNCTION_BLOCK "FB23_RA_AI_CUSTOM"   // FB23, LAD
{ S7_Optimized_Access := 'TRUE' }
VERSION : 0.1
   VAR_INPUT
      IN0 : Bool;
      IN1 : Bool;
      IN2 : Int;
      IN3 : Real;
      IN4 : Real;
      IN5 : Real;
      IN6 : Real;
      IN7 : Real;
      IN8 : Real;
      IN9 : Bool;
      IN10 : Bool;
      IN11 : Bool;
      IN12 : Bool;
      IN13 : Real;
      IN14 : Real;
   END_VAR
   VAR_OUTPUT
      Out15 : Real;
      Out16 : Bool;
      Out17 : Bool;
      Out18 : Bool;
      Out19 : Bool;
      Out20 : Bool;
   END_VAR
   VAR_IN_OUT
      IO21 : Real;
   END_VAR
   VAR_TEMP
      Temp22 : Word;
      INN2 : Int;
   END_VAR
BEGIN

REGION Network 1
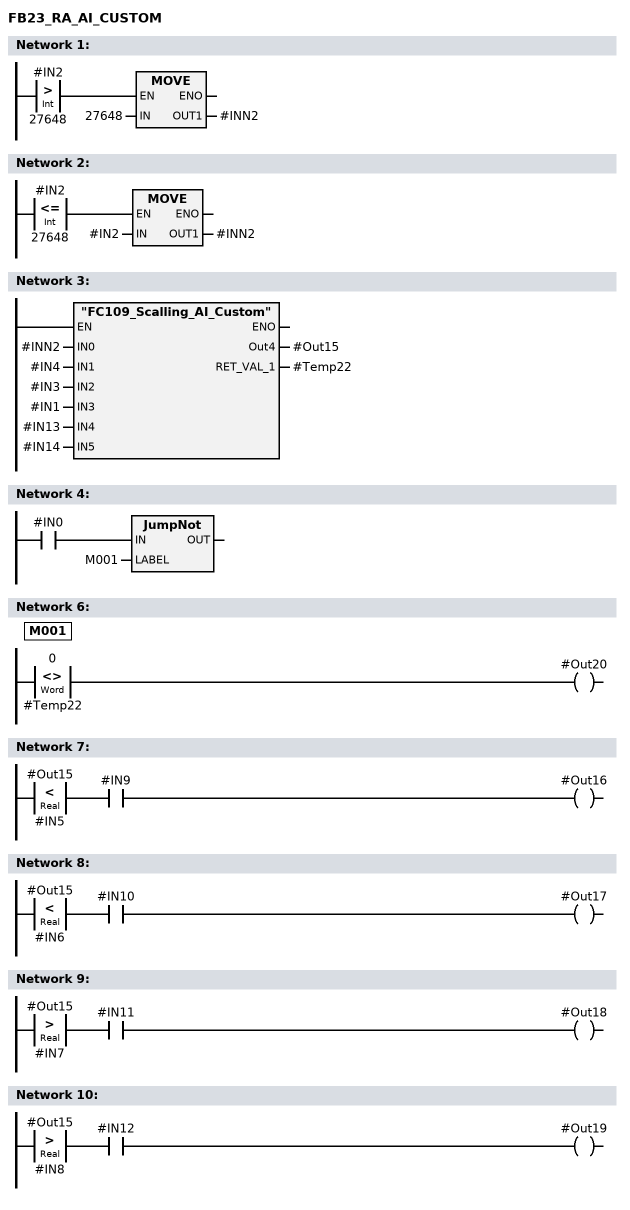
   RUNG wire#powerrail
      { S7_Templates := "SrcType := Int" } GT_Contact(in1 := #IN2, in2 := 27648)
      Move(in := 27648, out1 => #INN2)
   END_RUNG
   // the same network as SCL:
   IF #IN2 > 27648 THEN #INN2 := 27648; END_IF;
END_REGION

REGION Network 2
   RUNG wire#powerrail
      { S7_Templates := "SrcType := Int" } LE_Contact(in1 := #IN2, in2 := 27648)
      Move(in := #IN2, out1 => #INN2)
   END_RUNG
   // the same network as SCL:
   IF #IN2 <= 27648 THEN #INN2 := #IN2; END_IF;
END_REGION

REGION Network 3
   RUNG wire#powerrail
      "FC109_Scalling_AI_Custom"(IN0 := #INN2, IN1 := #IN4, IN2 := #IN3, IN3 := #IN1, IN4 := #IN13, IN5 := #IN14, Out4 => #Out15, RET_VAL_1 => #Temp22)
   END_RUNG
   // the same network as SCL:
   "FC109_Scalling_AI_Custom"(IN0 := #INN2,
                           IN1 := #IN4,
                           IN2 := #IN3,
                           IN3 := #IN1,
                           IN4 := #IN13,
                           IN5 := #IN14,
                           Out4 => #Out15,
                           RET_VAL_1 => #Temp22);
END_REGION

REGION Network 4
   // no SCL statement known for JumpNot: written as a call
   JumpNot(in := #IN0, label := M001);
END_REGION

REGION Network 6
   Label( M001 )
   RUNG wire#powerrail
      { S7_Templates := "SrcType := Word" } NE_Contact(in1 := 0, in2 := #Temp22)
      Coil( #Out20 )
   END_RUNG
   // the same network as SCL:
   M001:
   #Out20 := 0 <> #Temp22;
END_REGION

REGION Network 7
   RUNG wire#powerrail
      { S7_Templates := "SrcType := Real" } LT_Contact(in1 := #Out15, in2 := #IN5)
      Contact( #IN9 )
      Coil( #Out16 )
   END_RUNG
   // the same network as SCL:
   #Out16 := (#Out15 < #IN5) AND #IN9;
END_REGION

REGION Network 8
   RUNG wire#powerrail
      { S7_Templates := "SrcType := Real" } LT_Contact(in1 := #Out15, in2 := #IN6)
      Contact( #IN10 )
      Coil( #Out17 )
   END_RUNG
   // the same network as SCL:
   #Out17 := (#Out15 < #IN6) AND #IN10;
END_REGION

REGION Network 9
   RUNG wire#powerrail
      { S7_Templates := "SrcType := Real" } GT_Contact(in1 := #Out15, in2 := #IN7)
      Contact( #IN11 )
      Coil( #Out18 )
   END_RUNG
   // the same network as SCL:
   #Out18 := (#Out15 > #IN7) AND #IN11;
END_REGION

REGION Network 10
   RUNG wire#powerrail
      { S7_Templates := "SrcType := Real" } GT_Contact(in1 := #Out15, in2 := #IN8)
      Contact( #IN12 )
      Coil( #Out19 )
   END_RUNG
   // the same network as SCL:
   #Out19 := (#Out15 > #IN8) AND #IN12;
END_REGION
END_FUNCTION_BLOCK

FUNCTION "FC1_FEED_PUMPS" : Void   // FC1, LAD
TITLE = FEED PUMPS OPERATION
{ S7_Optimized_Access := 'TRUE' }
VERSION : 0.1
// FEED PUMP 1 = I 2.2
// FEED PUMP 2 = I 2.3
// 
// AO FEED PUMP 1 = QW 500
// AO FEED PUMP 2 = QW 502
// 
// AI FEED PUMP 1 = IW 106
// AI FEED PUMP 2 = IW 108
   VAR_TEMP
      Out1 : DInt;
      Out2 : Real;
      Out3 : DInt;
      Out4 : Real;
   END_VAR
   VAR_TEMP   // added for the SCL form of the ladder/FBD networks
      _w1 : Bool;
      _w2 : Bool;
   END_VAR
BEGIN

REGION Network 1: MOVE PARAMETER PID FROM HMI
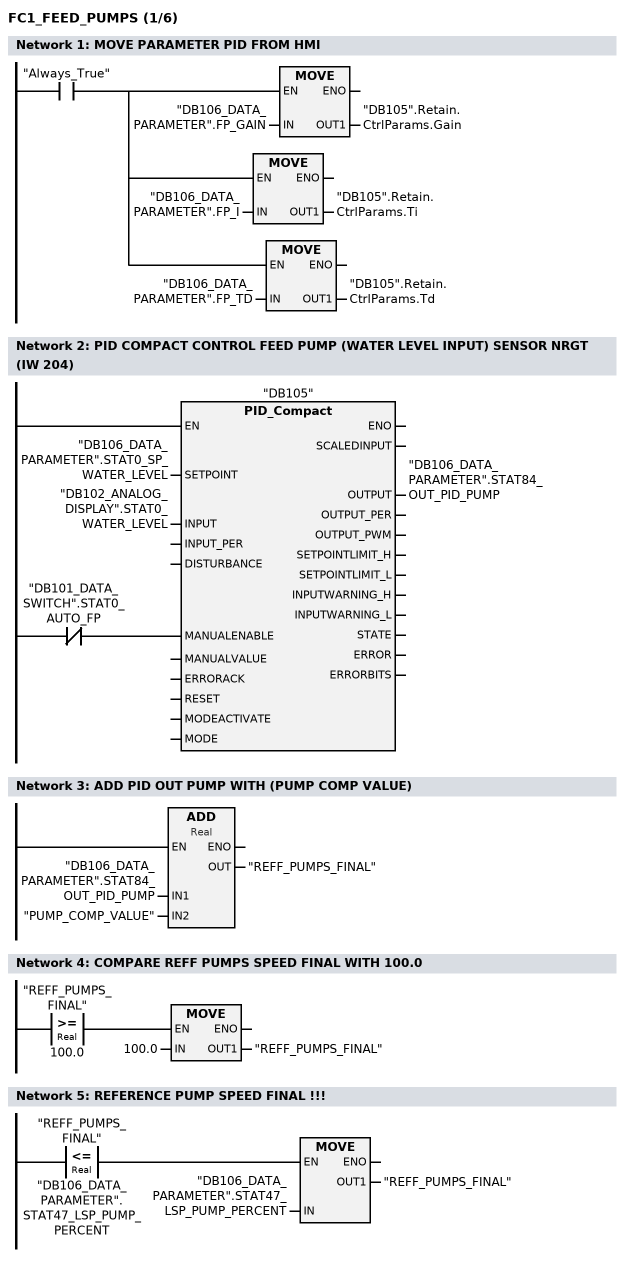
   RUNG wire#powerrail
      Contact( "Always_True" )
      wire#w1
      Move(in := "DB106_DATA_PARAMETER".FP_GAIN, out1 => "DB105".Retain.CtrlParams.Gain)
   END_RUNG
   RUNG wire#w1
      Move(in := "DB106_DATA_PARAMETER".FP_I, out1 => "DB105".Retain.CtrlParams.Ti)
   END_RUNG
   RUNG wire#w1
      Move(in := "DB106_DATA_PARAMETER".FP_TD, out1 => "DB105".Retain.CtrlParams.Td)
   END_RUNG
   // the same network as SCL:
   IF "Always_True" THEN
       "DB105".Retain.CtrlParams.Gain := "DB106_DATA_PARAMETER".FP_GAIN;
       "DB105".Retain.CtrlParams.Ti := "DB106_DATA_PARAMETER".FP_I;
       "DB105".Retain.CtrlParams.Td := "DB106_DATA_PARAMETER".FP_TD;
   END_IF;
END_REGION

REGION Network 2: PID COMPACT CONTROL FEED PUMP (WATER LEVEL INPUT) SENSOR NRGT (IW 204)
   "DB105"(Setpoint := "DB106_DATA_PARAMETER".STAT0_SP_WATER_LEVEL,   // PID_Compact
           Input := "DB102_ANALOG_DISPLAY".STAT0_WATER_LEVEL,
           ManualEnable := NOT "DB101_DATA_SWITCH".STAT0_AUTO_FP,
           Output => "DB106_DATA_PARAMETER".STAT84_OUT_PID_PUMP);
END_REGION

REGION Network 3: ADD PID OUT PUMP WITH (PUMP COMP VALUE)
   RUNG wire#powerrail
      { S7_Templates := "SrcType := Real" } Add(in1 := "DB106_DATA_PARAMETER".STAT84_OUT_PID_PUMP, in2 := "PUMP_COMP_VALUE", out => "REFF_PUMPS_FINAL")
   END_RUNG
   // the same network as SCL:
   "REFF_PUMPS_FINAL" := "DB106_DATA_PARAMETER".STAT84_OUT_PID_PUMP + "PUMP_COMP_VALUE";
END_REGION

REGION Network 4: COMPARE REFF PUMPS SPEED FINAL WITH 100.0
   RUNG wire#powerrail
      { S7_Templates := "SrcType := Real" } GE_Contact(in1 := "REFF_PUMPS_FINAL", in2 := 100.0)
      Move(in := 100.0, out1 => "REFF_PUMPS_FINAL")
   END_RUNG
   // the same network as SCL:
   IF "REFF_PUMPS_FINAL" >= 100.0 THEN "REFF_PUMPS_FINAL" := 100.0; END_IF;
END_REGION

REGION Network 5: REFERENCE PUMP SPEED FINAL !!!
   RUNG wire#powerrail
      { S7_Templates := "SrcType := Real" } LE_Contact(in1 := "REFF_PUMPS_FINAL", in2 := "DB106_DATA_PARAMETER".STAT47_LSP_PUMP_PERCENT)
      Move(in := "DB106_DATA_PARAMETER".STAT47_LSP_PUMP_PERCENT, out1 => "REFF_PUMPS_FINAL")
   END_RUNG
   // the same network as SCL:
   IF "REFF_PUMPS_FINAL" <= "DB106_DATA_PARAMETER".STAT47_LSP_PUMP_PERCENT THEN
       "REFF_PUMPS_FINAL" := "DB106_DATA_PARAMETER".STAT47_LSP_PUMP_PERCENT;
   END_IF;
END_REGION

REGION Network 6: SCALLING FEED PUMP 1 REFERENCE SPEED AO
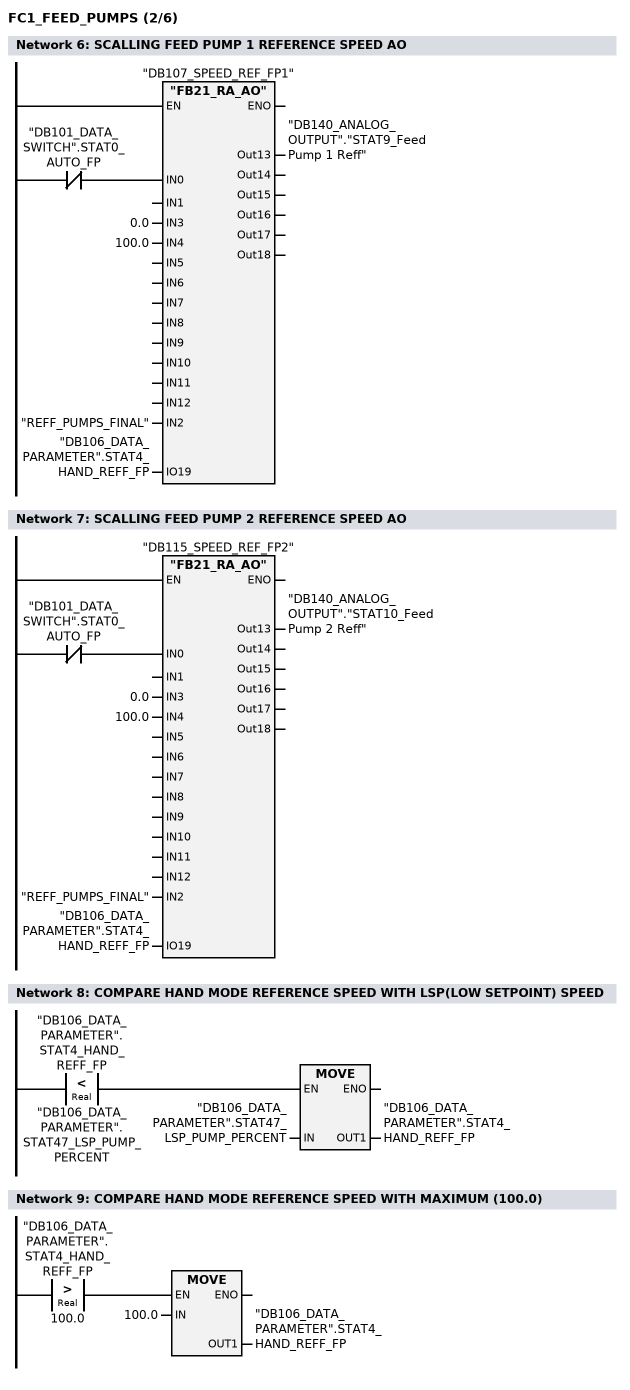
   RUNG wire#powerrail
      "DB107_SPEED_REF_FP1"(IN0 := wire#w1, IN1 :=, IN3 := 0.0, IN4 := 100.0, IN5 :=, IN6 :=, IN7 :=, IN8 :=, IN9 :=, IN10 :=, IN11 :=, IN12 :=, IN2 := "REFF_PUMPS_FINAL", IO19 := "DB106_DATA_PARAMETER".STAT4_HAND_REFF_FP, Out13 => "DB140_ANALOG_OUTPUT"."STAT9_Feed Pump 1 Reff", Out14 =>, Out15 =>, Out16 =>, Out17 =>, Out18 =>)
   END_RUNG
   RUNG wire#powerrail
      I_Contact( "DB101_DATA_SWITCH".STAT0_AUTO_FP )
   END_RUNG wire#w1
   // the same network as SCL:
   "DB107_SPEED_REF_FP1"(IN0 := NOT "DB101_DATA_SWITCH".STAT0_AUTO_FP,   // "FB21_RA_AO"
                         IN3 := 0.0,
                         IN4 := 100.0,
                         IN2 := "REFF_PUMPS_FINAL",
                         IO19 := "DB106_DATA_PARAMETER".STAT4_HAND_REFF_FP,
                         Out13 => "DB140_ANALOG_OUTPUT"."STAT9_Feed Pump 1 Reff");
END_REGION

REGION Network 7: SCALLING FEED PUMP 2 REFERENCE SPEED AO
   RUNG wire#powerrail
      "DB115_SPEED_REF_FP2"(IN0 := wire#w1, IN1 :=, IN3 := 0.0, IN4 := 100.0, IN5 :=, IN6 :=, IN7 :=, IN8 :=, IN9 :=, IN10 :=, IN11 :=, IN12 :=, IN2 := "REFF_PUMPS_FINAL", IO19 := "DB106_DATA_PARAMETER".STAT4_HAND_REFF_FP, Out13 => "DB140_ANALOG_OUTPUT"."STAT10_Feed Pump 2 Reff", Out14 =>, Out15 =>, Out16 =>, Out17 =>, Out18 =>)
   END_RUNG
   RUNG wire#powerrail
      I_Contact( "DB101_DATA_SWITCH".STAT0_AUTO_FP )
   END_RUNG wire#w1
   // the same network as SCL:
   "DB115_SPEED_REF_FP2"(IN0 := NOT "DB101_DATA_SWITCH".STAT0_AUTO_FP,   // "FB21_RA_AO"
                         IN3 := 0.0,
                         IN4 := 100.0,
                         IN2 := "REFF_PUMPS_FINAL",
                         IO19 := "DB106_DATA_PARAMETER".STAT4_HAND_REFF_FP,
                         Out13 => "DB140_ANALOG_OUTPUT"."STAT10_Feed Pump 2 Reff");
END_REGION

REGION Network 8: COMPARE HAND MODE REFERENCE SPEED WITH LSP(LOW SETPOINT) SPEED
   RUNG wire#powerrail
      { S7_Templates := "SrcType := Real" } LT_Contact(in1 := "DB106_DATA_PARAMETER".STAT4_HAND_REFF_FP, in2 := "DB106_DATA_PARAMETER".STAT47_LSP_PUMP_PERCENT)
      Move(in := "DB106_DATA_PARAMETER".STAT47_LSP_PUMP_PERCENT, out1 => "DB106_DATA_PARAMETER".STAT4_HAND_REFF_FP)
   END_RUNG
   // the same network as SCL:
   IF "DB106_DATA_PARAMETER".STAT4_HAND_REFF_FP < "DB106_DATA_PARAMETER".STAT47_LSP_PUMP_PERCENT THEN
       "DB106_DATA_PARAMETER".STAT4_HAND_REFF_FP := "DB106_DATA_PARAMETER".STAT47_LSP_PUMP_PERCENT;
   END_IF;
END_REGION

REGION Network 9: COMPARE HAND MODE REFERENCE SPEED WITH MAXIMUM (100.0)
   RUNG wire#powerrail
      { S7_Templates := "SrcType := Real" } GT_Contact(in1 := "DB106_DATA_PARAMETER".STAT4_HAND_REFF_FP, in2 := 100.0)
      Move(in := 100.0, out1 => "DB106_DATA_PARAMETER".STAT4_HAND_REFF_FP)
   END_RUNG
   // the same network as SCL:
   IF "DB106_DATA_PARAMETER".STAT4_HAND_REFF_FP > 100.0 THEN
       "DB106_DATA_PARAMETER".STAT4_HAND_REFF_FP := 100.0;
   END_IF;
END_REGION

REGION Network 10: HAND MODE SPEED UP FEED PUMP
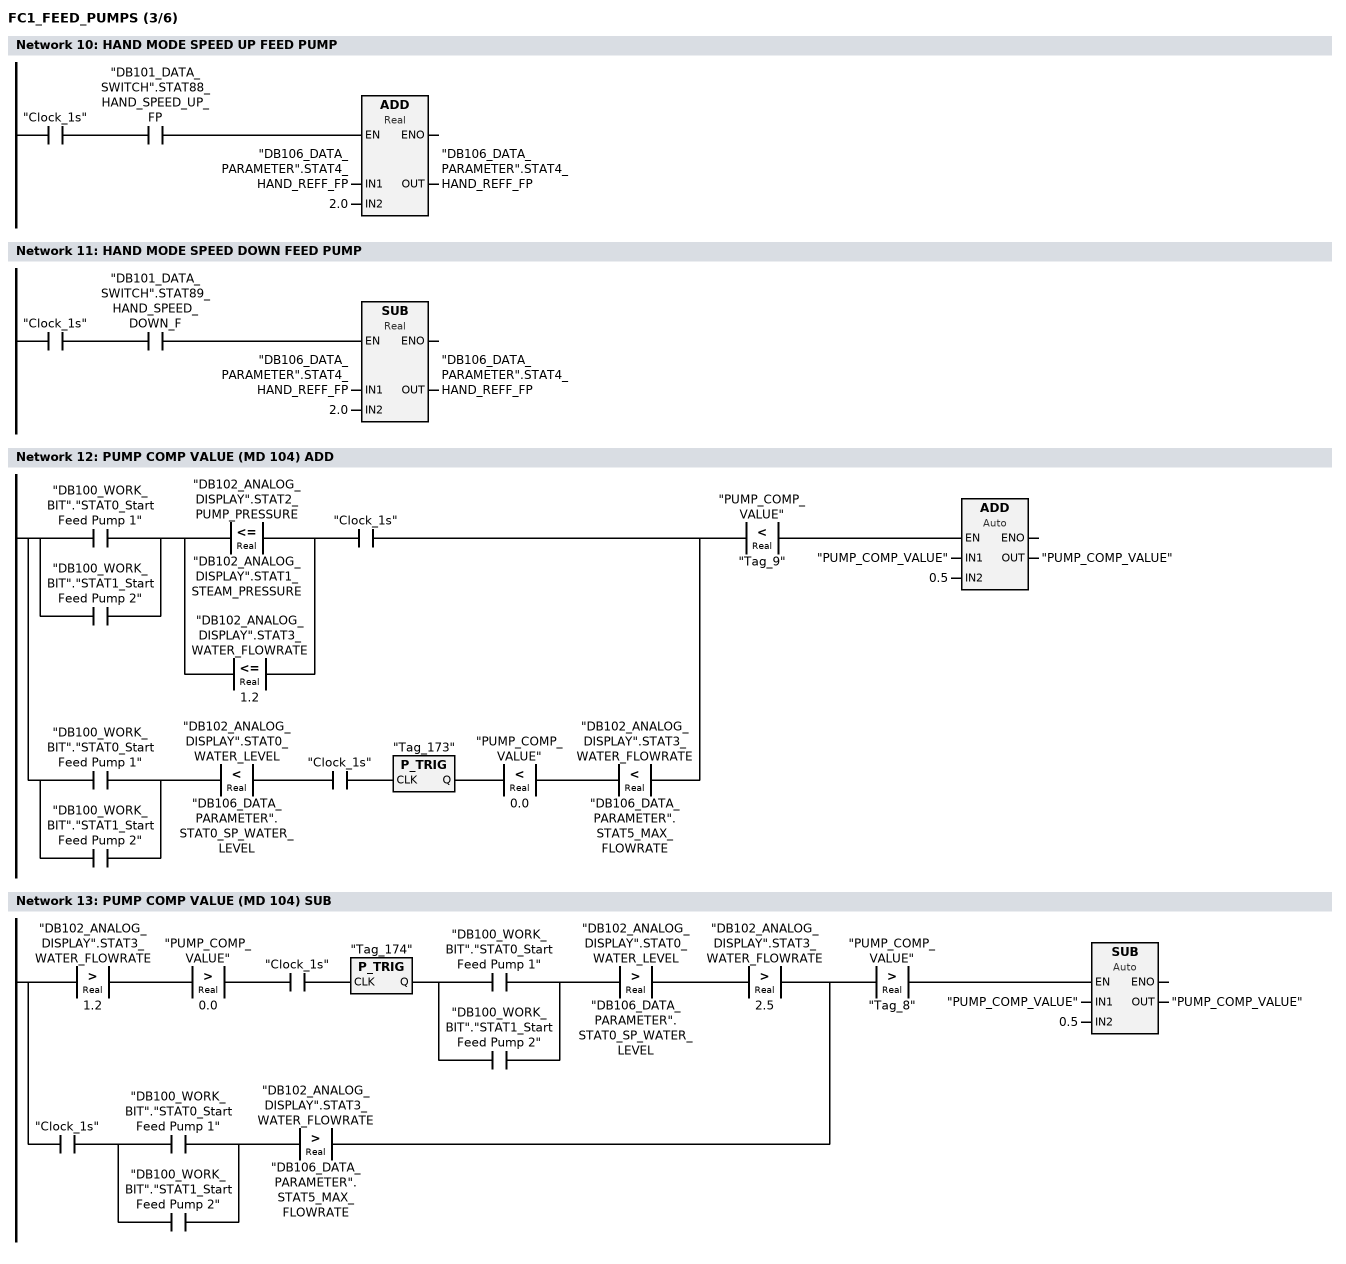
   RUNG wire#powerrail
      Contact( "Clock_1s" )
      Contact( "DB101_DATA_SWITCH".STAT88_HAND_SPEED_UP_FP )
      { S7_Templates := "SrcType := Real" } Add(in1 := "DB106_DATA_PARAMETER".STAT4_HAND_REFF_FP, in2 := 2.0, out => "DB106_DATA_PARAMETER".STAT4_HAND_REFF_FP)
   END_RUNG
   // the same network as SCL:
   IF "Clock_1s" AND "DB101_DATA_SWITCH".STAT88_HAND_SPEED_UP_FP THEN
       "DB106_DATA_PARAMETER".STAT4_HAND_REFF_FP := "DB106_DATA_PARAMETER".STAT4_HAND_REFF_FP + 2.0;
   END_IF;
END_REGION

REGION Network 11: HAND MODE SPEED DOWN FEED PUMP
   RUNG wire#powerrail
      Contact( "Clock_1s" )
      Contact( "DB101_DATA_SWITCH".STAT89_HAND_SPEED_DOWN_F )
      { S7_Templates := "SrcType := Real" } Sub(in1 := "DB106_DATA_PARAMETER".STAT4_HAND_REFF_FP, in2 := 2.0, out => "DB106_DATA_PARAMETER".STAT4_HAND_REFF_FP)
   END_RUNG
   // the same network as SCL:
   IF "Clock_1s" AND "DB101_DATA_SWITCH".STAT89_HAND_SPEED_DOWN_F THEN
       "DB106_DATA_PARAMETER".STAT4_HAND_REFF_FP := "DB106_DATA_PARAMETER".STAT4_HAND_REFF_FP - 2.0;
   END_IF;
END_REGION

REGION Network 12: PUMP COMP VALUE (MD 104) ADD
   RUNG wire#powerrail
      Contact( "DB100_WORK_BIT"."STAT0_Start Feed Pump 1" )
      wire#w1
      { S7_Templates := "SrcType := Real" } LE_Contact(in1 := "DB102_ANALOG_DISPLAY".STAT2_PUMP_PRESSURE, in2 := "DB102_ANALOG_DISPLAY".STAT1_STEAM_PRESSURE)
      wire#w2
      Contact( "Clock_1s" )
      wire#w3
      { S7_Templates := "SrcType := Real" } LT_Contact(in1 := "PUMP_COMP_VALUE", in2 := "Tag_9")
      Add(in1 := "PUMP_COMP_VALUE", in2 := 0.5, out => "PUMP_COMP_VALUE")
   END_RUNG
   RUNG wire#powerrail
      Contact( "DB100_WORK_BIT"."STAT1_Start Feed Pump 2" )
   END_RUNG wire#w1
   RUNG wire#w1
      { S7_Templates := "SrcType := Real" } LE_Contact(in1 := "DB102_ANALOG_DISPLAY".STAT3_WATER_FLOWRATE, in2 := 1.2)
   END_RUNG wire#w2
   RUNG wire#powerrail
      Contact( "DB100_WORK_BIT"."STAT0_Start Feed Pump 1" )
      wire#w4
      { S7_Templates := "SrcType := Real" } LT_Contact(in1 := "DB102_ANALOG_DISPLAY".STAT0_WATER_LEVEL, in2 := "DB106_DATA_PARAMETER".STAT0_SP_WATER_LEVEL)
      Contact( "Clock_1s" )
      P_Trig( "Tag_173" )
      { S7_Templates := "SrcType := Real" } LT_Contact(in1 := "PUMP_COMP_VALUE", in2 := 0.0)
      { S7_Templates := "SrcType := Real" } LT_Contact(in1 := "DB102_ANALOG_DISPLAY".STAT3_WATER_FLOWRATE, in2 := "DB106_DATA_PARAMETER".STAT5_MAX_FLOWRATE)
   END_RUNG wire#w3
   RUNG wire#powerrail
      Contact( "DB100_WORK_BIT"."STAT1_Start Feed Pump 2" )
   END_RUNG wire#w4
   // the same network as SCL:
   #_w1 := ("DB100_WORK_BIT"."STAT0_Start Feed Pump 1" OR "DB100_WORK_BIT"."STAT1_Start Feed Pump 2") AND ("DB102_ANALOG_DISPLAY".STAT0_WATER_LEVEL < "DB106_DATA_PARAMETER".STAT0_SP_WATER_LEVEL) AND "Clock_1s";
   #_w2 := #_w1 AND NOT "Tag_173";   // rising edge
   "Tag_173" := #_w1;
   IF ((("DB100_WORK_BIT"."STAT0_Start Feed Pump 1" OR "DB100_WORK_BIT"."STAT1_Start Feed Pump 2") AND (("DB102_ANALOG_DISPLAY".STAT2_PUMP_PRESSURE <= "DB102_ANALOG_DISPLAY".STAT1_STEAM_PRESSURE) OR ("DB102_ANALOG_DISPLAY".STAT3_WATER_FLOWRATE <= 1.2)) AND "Clock_1s") OR (#_w2 AND ("PUMP_COMP_VALUE" < 0.0) AND ("DB102_ANALOG_DISPLAY".STAT3_WATER_FLOWRATE < "DB106_DATA_PARAMETER".STAT5_MAX_FLOWRATE))) AND ("PUMP_COMP_VALUE" < "Tag_9") THEN
       "PUMP_COMP_VALUE" := "PUMP_COMP_VALUE" + 0.5;
   END_IF;
END_REGION

REGION Network 13: PUMP COMP VALUE (MD 104) SUB
   RUNG wire#powerrail
      { S7_Templates := "SrcType := Real" } GT_Contact(in1 := "DB102_ANALOG_DISPLAY".STAT3_WATER_FLOWRATE, in2 := 1.2)
      { S7_Templates := "SrcType := Real" } GT_Contact(in1 := "PUMP_COMP_VALUE", in2 := 0.0)
      Contact( "Clock_1s" )
      P_Trig( "Tag_174" )
      wire#w1
      Contact( "DB100_WORK_BIT"."STAT0_Start Feed Pump 1" )
      wire#w2
      { S7_Templates := "SrcType := Real" } GT_Contact(in1 := "DB102_ANALOG_DISPLAY".STAT0_WATER_LEVEL, in2 := "DB106_DATA_PARAMETER".STAT0_SP_WATER_LEVEL)
      { S7_Templates := "SrcType := Real" } GT_Contact(in1 := "DB102_ANALOG_DISPLAY".STAT3_WATER_FLOWRATE, in2 := 2.5)
      wire#w3
      { S7_Templates := "SrcType := Real" } GT_Contact(in1 := "PUMP_COMP_VALUE", in2 := "Tag_8")
      Sub(in1 := "PUMP_COMP_VALUE", in2 := 0.5, out => "PUMP_COMP_VALUE")
   END_RUNG
   RUNG wire#w1
      Contact( "DB100_WORK_BIT"."STAT1_Start Feed Pump 2" )
   END_RUNG wire#w2
   RUNG wire#powerrail
      Contact( "Clock_1s" )
      wire#w4
      Contact( "DB100_WORK_BIT"."STAT0_Start Feed Pump 1" )
      wire#w5
      { S7_Templates := "SrcType := Real" } GT_Contact(in1 := "DB102_ANALOG_DISPLAY".STAT3_WATER_FLOWRATE, in2 := "DB106_DATA_PARAMETER".STAT5_MAX_FLOWRATE)
   END_RUNG wire#w3
   RUNG wire#w4
      Contact( "DB100_WORK_BIT"."STAT1_Start Feed Pump 2" )
   END_RUNG wire#w5
   // the same network as SCL:
   #_w1 := ("DB102_ANALOG_DISPLAY".STAT3_WATER_FLOWRATE > 1.2) AND ("PUMP_COMP_VALUE" > 0.0) AND "Clock_1s";
   #_w2 := #_w1 AND NOT "Tag_174";   // rising edge
   "Tag_174" := #_w1;
   IF ((#_w2 AND ("DB100_WORK_BIT"."STAT0_Start Feed Pump 1" OR "DB100_WORK_BIT"."STAT1_Start Feed Pump 2") AND ("DB102_ANALOG_DISPLAY".STAT0_WATER_LEVEL > "DB106_DATA_PARAMETER".STAT0_SP_WATER_LEVEL) AND ("DB102_ANALOG_DISPLAY".STAT3_WATER_FLOWRATE > 2.5)) OR ("Clock_1s" AND ("DB100_WORK_BIT"."STAT0_Start Feed Pump 1" OR "DB100_WORK_BIT"."STAT1_Start Feed Pump 2") AND ("DB102_ANALOG_DISPLAY".STAT3_WATER_FLOWRATE > "DB106_DATA_PARAMETER".STAT5_MAX_FLOWRATE))) AND ("PUMP_COMP_VALUE" > "Tag_8") THEN
       "PUMP_COMP_VALUE" := "PUMP_COMP_VALUE" - 0.5;
   END_IF;
END_REGION

REGION Network 14: Network 13
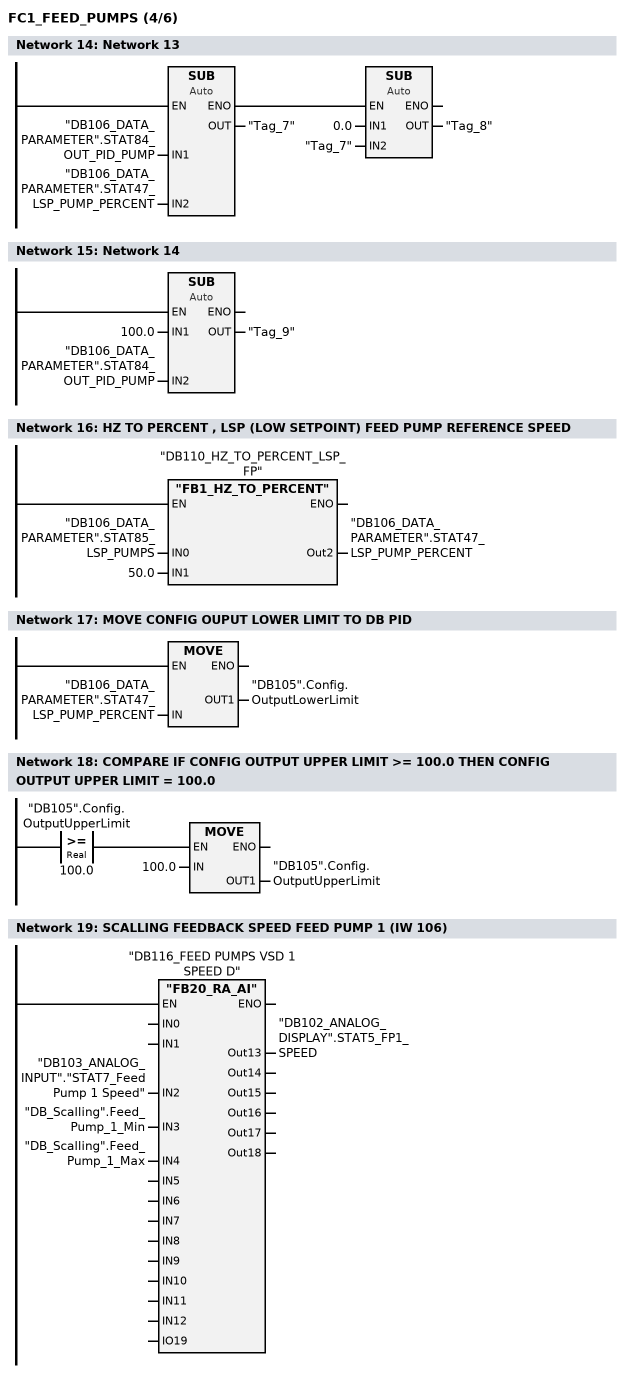
   RUNG wire#powerrail
      Sub(in1 := "DB106_DATA_PARAMETER".STAT84_OUT_PID_PUMP, in2 := "DB106_DATA_PARAMETER".STAT47_LSP_PUMP_PERCENT, out => "Tag_7")
      Sub(in1 := 0.0, in2 := "Tag_7", out => "Tag_8")
   END_RUNG
   // the same network as SCL:
   "Tag_7" := "DB106_DATA_PARAMETER".STAT84_OUT_PID_PUMP - "DB106_DATA_PARAMETER".STAT47_LSP_PUMP_PERCENT;
   "Tag_8" := 0.0 - "Tag_7";
END_REGION

REGION Network 15: Network 14
   RUNG wire#powerrail
      Sub(in1 := 100.0, in2 := "DB106_DATA_PARAMETER".STAT84_OUT_PID_PUMP, out => "Tag_9")
   END_RUNG
   // the same network as SCL:
   "Tag_9" := 100.0 - "DB106_DATA_PARAMETER".STAT84_OUT_PID_PUMP;
END_REGION

REGION Network 16: HZ TO PERCENT , LSP (LOW SETPOINT) FEED PUMP REFERENCE SPEED
   RUNG wire#powerrail
      "DB110_HZ_TO_PERCENT_LSP_FP"(IN0 := "DB106_DATA_PARAMETER".STAT85_LSP_PUMPS, IN1 := 50.0, Out2 => "DB106_DATA_PARAMETER".STAT47_LSP_PUMP_PERCENT)
   END_RUNG
   // the same network as SCL:
   "DB110_HZ_TO_PERCENT_LSP_FP"(IN0 := "DB106_DATA_PARAMETER".STAT85_LSP_PUMPS,   // "FB1_HZ_TO_PERCENT"
                           IN1 := 50.0,
                           Out2 => "DB106_DATA_PARAMETER".STAT47_LSP_PUMP_PERCENT);
END_REGION

REGION Network 17: MOVE CONFIG OUPUT LOWER LIMIT TO DB PID
   RUNG wire#powerrail
      Move(in := "DB106_DATA_PARAMETER".STAT47_LSP_PUMP_PERCENT, out1 => "DB105".Config.OutputLowerLimit)
   END_RUNG
   // the same network as SCL:
   "DB105".Config.OutputLowerLimit := "DB106_DATA_PARAMETER".STAT47_LSP_PUMP_PERCENT;
END_REGION

REGION Network 18: COMPARE IF CONFIG OUTPUT UPPER LIMIT >= 100.0 THEN CONFIG OUTPUT UPPER LIMIT = 100.0
   RUNG wire#powerrail
      { S7_Templates := "SrcType := Real" } GE_Contact(in1 := "DB105".Config.OutputUpperLimit, in2 := 100.0)
      Move(in := 100.0, out1 => "DB105".Config.OutputUpperLimit)
   END_RUNG
   // the same network as SCL:
   IF "DB105".Config.OutputUpperLimit >= 100.0 THEN "DB105".Config.OutputUpperLimit := 100.0; END_IF;
END_REGION

REGION Network 19: SCALLING FEEDBACK SPEED FEED PUMP 1 (IW 106)
   RUNG wire#powerrail
      "DB116_FEED PUMPS VSD 1 SPEED D"(IN0 :=, IN1 :=, IN2 := "DB103_ANALOG_INPUT"."STAT7_Feed Pump 1 Speed", IN3 := "DB_Scalling".Feed_Pump_1_Min, IN4 := "DB_Scalling".Feed_Pump_1_Max, IN5 :=, IN6 :=, IN7 :=, IN8 :=, IN9 :=, IN10 :=, IN11 :=, IN12 :=, IO19 :=, Out13 => "DB102_ANALOG_DISPLAY".STAT5_FP1_SPEED, Out14 =>, Out15 =>, Out16 =>, Out17 =>, Out18 =>)
   END_RUNG
   // the same network as SCL:
   "DB116_FEED PUMPS VSD 1 SPEED D"(IN2 := "DB103_ANALOG_INPUT"."STAT7_Feed Pump 1 Speed",   // "FB20_RA_AI"
                           IN3 := "DB_Scalling".Feed_Pump_1_Min,
                           IN4 := "DB_Scalling".Feed_Pump_1_Max,
                           Out13 => "DB102_ANALOG_DISPLAY".STAT5_FP1_SPEED);
END_REGION

REGION Network 20: SCALLING FEEDBACK SPEED FEED PUMP 2 (IW 108)
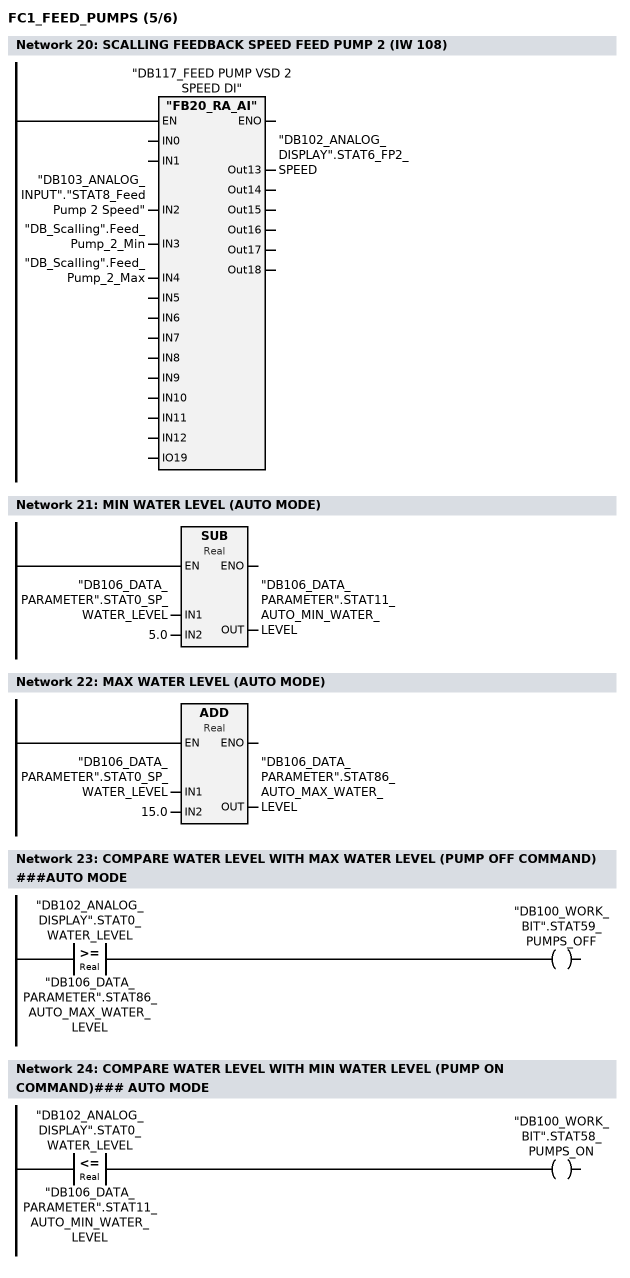
   RUNG wire#powerrail
      "DB117_FEED PUMP VSD 2 SPEED DI"(IN0 :=, IN1 :=, IN2 := "DB103_ANALOG_INPUT"."STAT8_Feed Pump 2 Speed", IN3 := "DB_Scalling".Feed_Pump_2_Min, IN4 := "DB_Scalling".Feed_Pump_2_Max, IN5 :=, IN6 :=, IN7 :=, IN8 :=, IN9 :=, IN10 :=, IN11 :=, IN12 :=, IO19 :=, Out13 => "DB102_ANALOG_DISPLAY".STAT6_FP2_SPEED, Out14 =>, Out15 =>, Out16 =>, Out17 =>, Out18 =>)
   END_RUNG
   // the same network as SCL:
   "DB117_FEED PUMP VSD 2 SPEED DI"(IN2 := "DB103_ANALOG_INPUT"."STAT8_Feed Pump 2 Speed",   // "FB20_RA_AI"
                           IN3 := "DB_Scalling".Feed_Pump_2_Min,
                           IN4 := "DB_Scalling".Feed_Pump_2_Max,
                           Out13 => "DB102_ANALOG_DISPLAY".STAT6_FP2_SPEED);
END_REGION

REGION Network 21: MIN WATER LEVEL (AUTO MODE)
   RUNG wire#powerrail
      { S7_Templates := "SrcType := Real" } Sub(in1 := "DB106_DATA_PARAMETER".STAT0_SP_WATER_LEVEL, in2 := 5.0, out => "DB106_DATA_PARAMETER".STAT11_AUTO_MIN_WATER_LEVEL)
   END_RUNG
   // the same network as SCL:
   "DB106_DATA_PARAMETER".STAT11_AUTO_MIN_WATER_LEVEL := "DB106_DATA_PARAMETER".STAT0_SP_WATER_LEVEL - 5.0;
END_REGION

REGION Network 22: MAX WATER LEVEL (AUTO MODE)
   RUNG wire#powerrail
      { S7_Templates := "SrcType := Real" } Add(in1 := "DB106_DATA_PARAMETER".STAT0_SP_WATER_LEVEL, in2 := 15.0, out => "DB106_DATA_PARAMETER".STAT86_AUTO_MAX_WATER_LEVEL)
   END_RUNG
   // the same network as SCL:
   "DB106_DATA_PARAMETER".STAT86_AUTO_MAX_WATER_LEVEL := "DB106_DATA_PARAMETER".STAT0_SP_WATER_LEVEL + 15.0;
END_REGION

REGION Network 23: COMPARE WATER LEVEL WITH MAX WATER LEVEL (PUMP OFF COMMAND) ###AUTO MODE
   RUNG wire#powerrail
      { S7_Templates := "SrcType := Real" } GE_Contact(in1 := "DB102_ANALOG_DISPLAY".STAT0_WATER_LEVEL, in2 := "DB106_DATA_PARAMETER".STAT86_AUTO_MAX_WATER_LEVEL)
      Coil( "DB100_WORK_BIT".STAT59_PUMPS_OFF )
   END_RUNG
   // the same network as SCL:
   "DB100_WORK_BIT".STAT59_PUMPS_OFF := "DB102_ANALOG_DISPLAY".STAT0_WATER_LEVEL >= "DB106_DATA_PARAMETER".STAT86_AUTO_MAX_WATER_LEVEL;
END_REGION

REGION Network 24: COMPARE WATER LEVEL WITH MIN WATER LEVEL (PUMP ON COMMAND)### AUTO MODE
   RUNG wire#powerrail
      { S7_Templates := "SrcType := Real" } LE_Contact(in1 := "DB102_ANALOG_DISPLAY".STAT0_WATER_LEVEL, in2 := "DB106_DATA_PARAMETER".STAT11_AUTO_MIN_WATER_LEVEL)
      Coil( "DB100_WORK_BIT".STAT58_PUMPS_ON )
   END_RUNG
   // the same network as SCL:
   "DB100_WORK_BIT".STAT58_PUMPS_ON := "DB102_ANALOG_DISPLAY".STAT0_WATER_LEVEL <= "DB106_DATA_PARAMETER".STAT11_AUTO_MIN_WATER_LEVEL;
END_REGION

REGION Network 25: PUMPS AUTOMATIC COMMAND
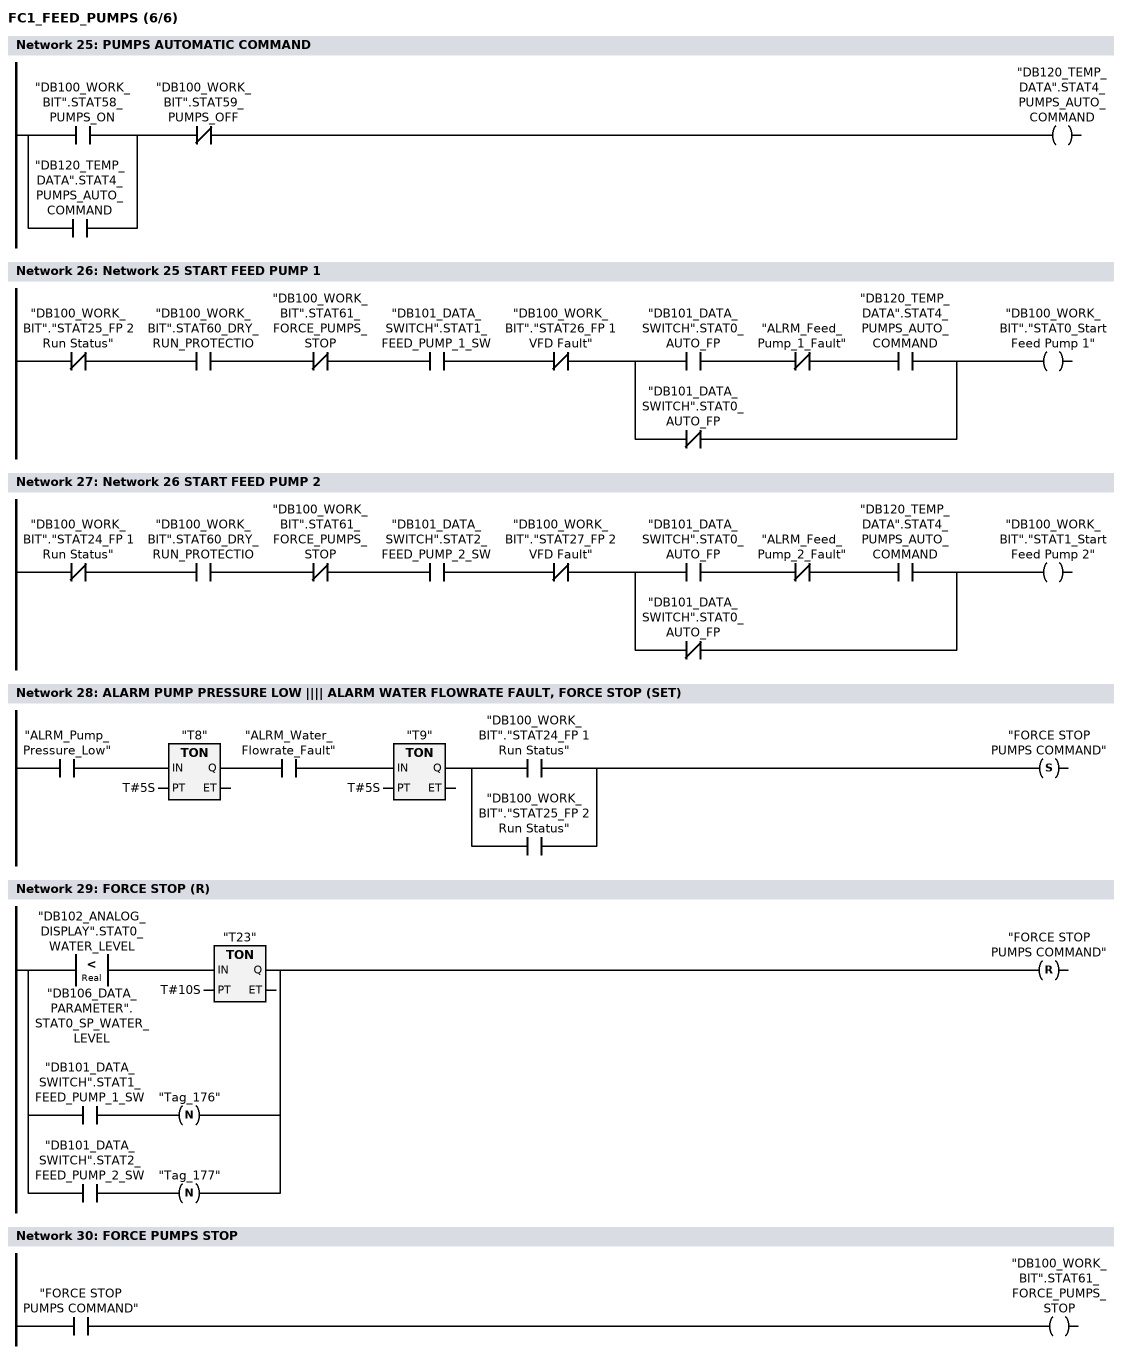
   RUNG wire#powerrail
      Contact( "DB100_WORK_BIT".STAT58_PUMPS_ON )
      wire#w1
      I_Contact( "DB100_WORK_BIT".STAT59_PUMPS_OFF )
      Coil( "DB120_TEMP_DATA".STAT4_PUMPS_AUTO_COMMAND )
   END_RUNG
   RUNG wire#powerrail
      Contact( "DB120_TEMP_DATA".STAT4_PUMPS_AUTO_COMMAND )
   END_RUNG wire#w1
   // the same network as SCL:
   "DB120_TEMP_DATA".STAT4_PUMPS_AUTO_COMMAND := ("DB100_WORK_BIT".STAT58_PUMPS_ON OR "DB120_TEMP_DATA".STAT4_PUMPS_AUTO_COMMAND) AND NOT "DB100_WORK_BIT".STAT59_PUMPS_OFF;
END_REGION

REGION Network 26: Network 25 START FEED PUMP 1
   RUNG wire#powerrail
      I_Contact( "DB100_WORK_BIT"."STAT25_FP 2 Run Status" )
      Contact( "DB100_WORK_BIT".STAT60_DRY_RUN_PROTECTIO )
      I_Contact( "DB100_WORK_BIT".STAT61_FORCE_PUMPS_STOP )
      Contact( "DB101_DATA_SWITCH".STAT1_FEED_PUMP_1_SW )
      I_Contact( "DB100_WORK_BIT"."STAT26_FP 1 VFD Fault" )
      wire#w1
      Contact( "DB101_DATA_SWITCH".STAT0_AUTO_FP )
      I_Contact( "ALRM_Feed_Pump_1_Fault" )
      Contact( "DB120_TEMP_DATA".STAT4_PUMPS_AUTO_COMMAND )
      wire#w2
      Coil( "DB100_WORK_BIT"."STAT0_Start Feed Pump 1" )
   END_RUNG
   RUNG wire#w1
      I_Contact( "DB101_DATA_SWITCH".STAT0_AUTO_FP )
   END_RUNG wire#w2
   // the same network as SCL:
   "DB100_WORK_BIT"."STAT0_Start Feed Pump 1" := NOT "DB100_WORK_BIT"."STAT25_FP 2 Run Status" AND "DB100_WORK_BIT".STAT60_DRY_RUN_PROTECTIO AND NOT "DB100_WORK_BIT".STAT61_FORCE_PUMPS_STOP AND "DB101_DATA_SWITCH".STAT1_FEED_PUMP_1_SW AND NOT "DB100_WORK_BIT"."STAT26_FP 1 VFD Fault" AND (("DB101_DATA_SWITCH".STAT0_AUTO_FP AND NOT "ALRM_Feed_Pump_1_Fault" AND "DB120_TEMP_DATA".STAT4_PUMPS_AUTO_COMMAND) OR NOT "DB101_DATA_SWITCH".STAT0_AUTO_FP);
END_REGION

REGION Network 27: Network 26 START FEED PUMP 2
   RUNG wire#powerrail
      I_Contact( "DB100_WORK_BIT"."STAT24_FP 1 Run Status" )
      Contact( "DB100_WORK_BIT".STAT60_DRY_RUN_PROTECTIO )
      I_Contact( "DB100_WORK_BIT".STAT61_FORCE_PUMPS_STOP )
      Contact( "DB101_DATA_SWITCH".STAT2_FEED_PUMP_2_SW )
      I_Contact( "DB100_WORK_BIT"."STAT27_FP 2 VFD Fault" )
      wire#w1
      Contact( "DB101_DATA_SWITCH".STAT0_AUTO_FP )
      I_Contact( "ALRM_Feed_Pump_2_Fault" )
      Contact( "DB120_TEMP_DATA".STAT4_PUMPS_AUTO_COMMAND )
      wire#w2
      Coil( "DB100_WORK_BIT"."STAT1_Start Feed Pump 2" )
   END_RUNG
   RUNG wire#w1
      I_Contact( "DB101_DATA_SWITCH".STAT0_AUTO_FP )
   END_RUNG wire#w2
   // the same network as SCL:
   "DB100_WORK_BIT"."STAT1_Start Feed Pump 2" := NOT "DB100_WORK_BIT"."STAT24_FP 1 Run Status" AND "DB100_WORK_BIT".STAT60_DRY_RUN_PROTECTIO AND NOT "DB100_WORK_BIT".STAT61_FORCE_PUMPS_STOP AND "DB101_DATA_SWITCH".STAT2_FEED_PUMP_2_SW AND NOT "DB100_WORK_BIT"."STAT27_FP 2 VFD Fault" AND (("DB101_DATA_SWITCH".STAT0_AUTO_FP AND NOT "ALRM_Feed_Pump_2_Fault" AND "DB120_TEMP_DATA".STAT4_PUMPS_AUTO_COMMAND) OR NOT "DB101_DATA_SWITCH".STAT0_AUTO_FP);
END_REGION

REGION Network 28: ALARM PUMP PRESSURE LOW |||| ALARM WATER FLOWRATE FAULT, FORCE STOP (SET)
   "T8".TON(IN := "ALRM_Pump_Pressure_Low", PT := T#5S);
   "T9".TON(IN := "T8".Q AND "ALRM_Water_Flowrate_Fault", PT := T#5S);
   IF "T9".Q AND ("DB100_WORK_BIT"."STAT24_FP 1 Run Status" OR "DB100_WORK_BIT"."STAT25_FP 2 Run Status") THEN
       "FORCE STOP PUMPS COMMAND" := TRUE;
   END_IF;
END_REGION

REGION Network 29: FORCE STOP (R)
   "T23".TON(IN := "DB102_ANALOG_DISPLAY".STAT0_WATER_LEVEL < "DB106_DATA_PARAMETER".STAT0_SP_WATER_LEVEL,
             PT := T#10S);
   #_w1 := NOT "DB101_DATA_SWITCH".STAT1_FEED_PUMP_1_SW AND "Tag_176";   // falling edge
   "Tag_176" := "DB101_DATA_SWITCH".STAT1_FEED_PUMP_1_SW;
   #_w2 := NOT "DB101_DATA_SWITCH".STAT2_FEED_PUMP_2_SW AND "Tag_177";   // falling edge
   "Tag_177" := "DB101_DATA_SWITCH".STAT2_FEED_PUMP_2_SW;
   IF "T23".Q OR #_w1 OR #_w2 THEN "FORCE STOP PUMPS COMMAND" := FALSE; END_IF;
END_REGION

REGION Network 30: FORCE PUMPS STOP
   RUNG wire#powerrail
      Contact( "FORCE STOP PUMPS COMMAND" )
      Coil( "DB100_WORK_BIT".STAT61_FORCE_PUMPS_STOP )
   END_RUNG
   // the same network as SCL:
   "DB100_WORK_BIT".STAT61_FORCE_PUMPS_STOP := "FORCE STOP PUMPS COMMAND";
END_REGION
END_FUNCTION

FUNCTION "FC2_scalling" : Void   // FC2, LAD
TITLE = SCALLING
{ S7_Optimized_Access := 'TRUE' }
VERSION : 0.1
BEGIN

REGION Network 1: Press Transducer | IW 100
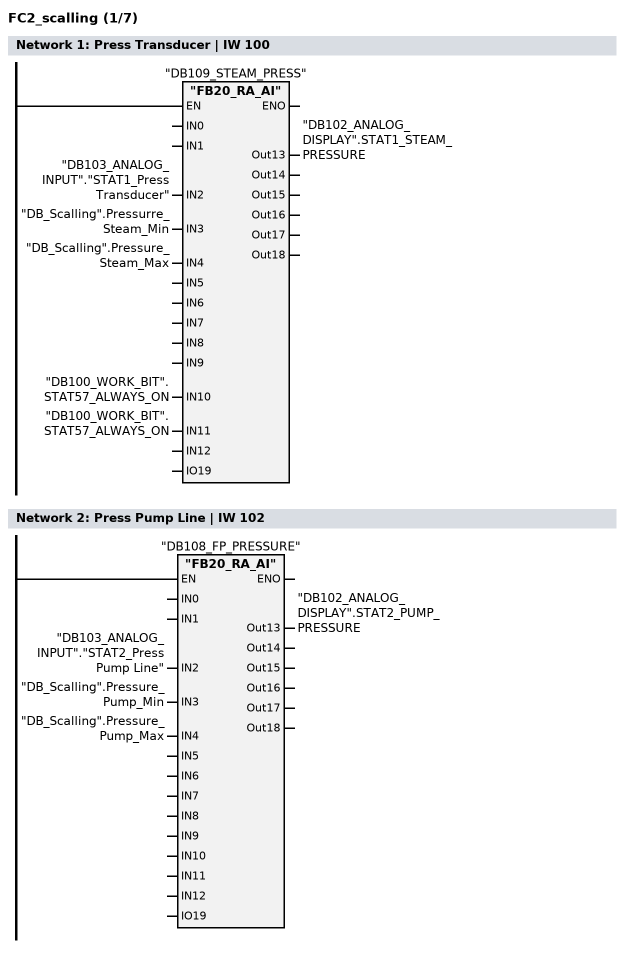
   RUNG wire#powerrail
      "DB109_STEAM_PRESS"(IN0 :=, IN1 :=, IN2 := "DB103_ANALOG_INPUT"."STAT1_Press Transducer", IN3 := "DB_Scalling".Pressurre_Steam_Min, IN4 := "DB_Scalling".Pressure_Steam_Max, IN5 :=, IN6 :=, IN7 :=, IN8 :=, IN9 :=, IN10 := "DB100_WORK_BIT".STAT57_ALWAYS_ON, IN11 := "DB100_WORK_BIT".STAT57_ALWAYS_ON, IN12 :=, IO19 :=, Out13 => "DB102_ANALOG_DISPLAY".STAT1_STEAM_PRESSURE, Out14 =>, Out15 =>, Out16 =>, Out17 =>, Out18 =>)
   END_RUNG
   // the same network as SCL:
   "DB109_STEAM_PRESS"(IN2 := "DB103_ANALOG_INPUT"."STAT1_Press Transducer",   // "FB20_RA_AI"
                       IN3 := "DB_Scalling".Pressurre_Steam_Min,
                       IN4 := "DB_Scalling".Pressure_Steam_Max,
                       IN10 := "DB100_WORK_BIT".STAT57_ALWAYS_ON,
                       IN11 := "DB100_WORK_BIT".STAT57_ALWAYS_ON,
                       Out13 => "DB102_ANALOG_DISPLAY".STAT1_STEAM_PRESSURE);
END_REGION

REGION Network 2: Press Pump Line | IW 102
   RUNG wire#powerrail
      "DB108_FP_PRESSURE"(IN0 :=, IN1 :=, IN2 := "DB103_ANALOG_INPUT"."STAT2_Press Pump Line", IN3 := "DB_Scalling".Pressure_Pump_Min, IN4 := "DB_Scalling".Pressure_Pump_Max, IN5 :=, IN6 :=, IN7 :=, IN8 :=, IN9 :=, IN10 :=, IN11 :=, IN12 :=, IO19 :=, Out13 => "DB102_ANALOG_DISPLAY".STAT2_PUMP_PRESSURE, Out14 =>, Out15 =>, Out16 =>, Out17 =>, Out18 =>)
   END_RUNG
   // the same network as SCL:
   "DB108_FP_PRESSURE"(IN2 := "DB103_ANALOG_INPUT"."STAT2_Press Pump Line",   // "FB20_RA_AI"
                       IN3 := "DB_Scalling".Pressure_Pump_Min,
                       IN4 := "DB_Scalling".Pressure_Pump_Max,
                       Out13 => "DB102_ANALOG_DISPLAY".STAT2_PUMP_PRESSURE);
END_REGION

REGION Network 3: NRGT (Level electrode) | IW 204
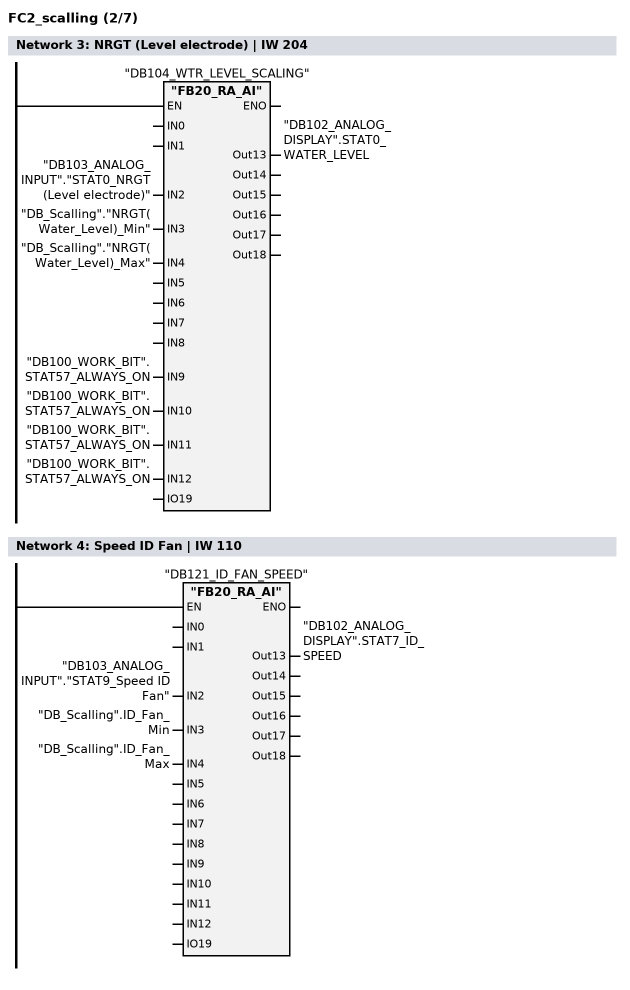
   RUNG wire#powerrail
      "DB104_WTR_LEVEL_SCALING"(IN0 :=, IN1 :=, IN2 := "DB103_ANALOG_INPUT"."STAT0_NRGT (Level electrode)", IN3 := "DB_Scalling"."NRGT(Water_Level)_Min", IN4 := "DB_Scalling"."NRGT(Water_Level)_Max", IN5 :=, IN6 :=, IN7 :=, IN8 :=, IN9 := "DB100_WORK_BIT".STAT57_ALWAYS_ON, IN10 := "DB100_WORK_BIT".STAT57_ALWAYS_ON, IN11 := "DB100_WORK_BIT".STAT57_ALWAYS_ON, IN12 := "DB100_WORK_BIT".STAT57_ALWAYS_ON, IO19 :=, Out13 => "DB102_ANALOG_DISPLAY".STAT0_WATER_LEVEL, Out14 =>, Out15 =>, Out16 =>, Out17 =>, Out18 =>)
   END_RUNG
   // the same network as SCL:
   "DB104_WTR_LEVEL_SCALING"(IN2 := "DB103_ANALOG_INPUT"."STAT0_NRGT (Level electrode)",   // "FB20_RA_AI"
                           IN3 := "DB_Scalling"."NRGT(Water_Level)_Min",
                           IN4 := "DB_Scalling"."NRGT(Water_Level)_Max",
                           IN9 := "DB100_WORK_BIT".STAT57_ALWAYS_ON,
                           IN10 := "DB100_WORK_BIT".STAT57_ALWAYS_ON,
                           IN11 := "DB100_WORK_BIT".STAT57_ALWAYS_ON,
                           IN12 := "DB100_WORK_BIT".STAT57_ALWAYS_ON,
                           Out13 => "DB102_ANALOG_DISPLAY".STAT0_WATER_LEVEL);
END_REGION

REGION Network 4: Speed ID Fan | IW 110
   RUNG wire#powerrail
      "DB121_ID_FAN_SPEED"(IN0 :=, IN1 :=, IN2 := "DB103_ANALOG_INPUT"."STAT9_Speed ID Fan", IN3 := "DB_Scalling".ID_Fan_Min, IN4 := "DB_Scalling".ID_Fan_Max, IN5 :=, IN6 :=, IN7 :=, IN8 :=, IN9 :=, IN10 :=, IN11 :=, IN12 :=, IO19 :=, Out13 => "DB102_ANALOG_DISPLAY".STAT7_ID_SPEED, Out14 =>, Out15 =>, Out16 =>, Out17 =>, Out18 =>)
   END_RUNG
   // the same network as SCL:
   "DB121_ID_FAN_SPEED"(IN2 := "DB103_ANALOG_INPUT"."STAT9_Speed ID Fan",   // "FB20_RA_AI"
                        IN3 := "DB_Scalling".ID_Fan_Min,
                        IN4 := "DB_Scalling".ID_Fan_Max,
                        Out13 => "DB102_ANALOG_DISPLAY".STAT7_ID_SPEED);
END_REGION

REGION Network 5: Speed LH FD Fan | IW 112
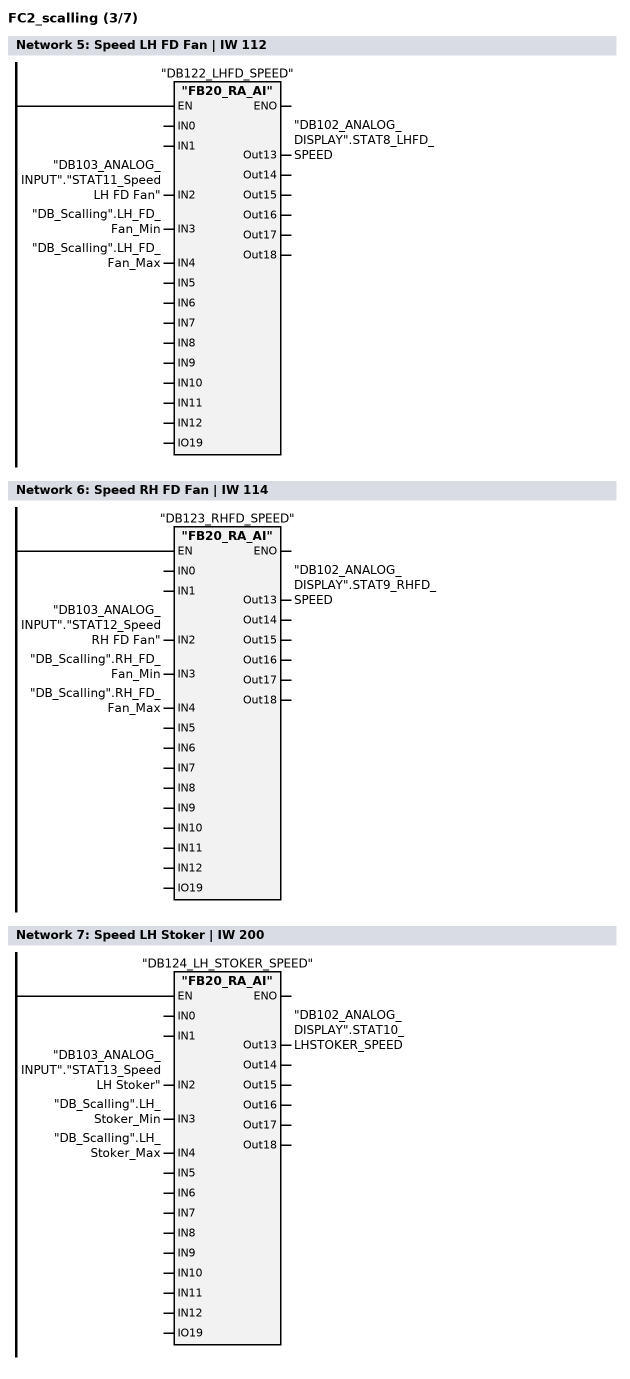
   RUNG wire#powerrail
      "DB122_LHFD_SPEED"(IN0 :=, IN1 :=, IN2 := "DB103_ANALOG_INPUT"."STAT11_Speed LH FD Fan", IN3 := "DB_Scalling".LH_FD_Fan_Min, IN4 := "DB_Scalling".LH_FD_Fan_Max, IN5 :=, IN6 :=, IN7 :=, IN8 :=, IN9 :=, IN10 :=, IN11 :=, IN12 :=, IO19 :=, Out13 => "DB102_ANALOG_DISPLAY".STAT8_LHFD_SPEED, Out14 =>, Out15 =>, Out16 =>, Out17 =>, Out18 =>)
   END_RUNG
   // the same network as SCL:
   "DB122_LHFD_SPEED"(IN2 := "DB103_ANALOG_INPUT"."STAT11_Speed LH FD Fan",   // "FB20_RA_AI"
                      IN3 := "DB_Scalling".LH_FD_Fan_Min,
                      IN4 := "DB_Scalling".LH_FD_Fan_Max,
                      Out13 => "DB102_ANALOG_DISPLAY".STAT8_LHFD_SPEED);
END_REGION

REGION Network 6: Speed RH FD Fan | IW 114
   RUNG wire#powerrail
      "DB123_RHFD_SPEED"(IN0 :=, IN1 :=, IN2 := "DB103_ANALOG_INPUT"."STAT12_Speed RH FD Fan", IN3 := "DB_Scalling".RH_FD_Fan_Min, IN4 := "DB_Scalling".RH_FD_Fan_Max, IN5 :=, IN6 :=, IN7 :=, IN8 :=, IN9 :=, IN10 :=, IN11 :=, IN12 :=, IO19 :=, Out13 => "DB102_ANALOG_DISPLAY".STAT9_RHFD_SPEED, Out14 =>, Out15 =>, Out16 =>, Out17 =>, Out18 =>)
   END_RUNG
   // the same network as SCL:
   "DB123_RHFD_SPEED"(IN2 := "DB103_ANALOG_INPUT"."STAT12_Speed RH FD Fan",   // "FB20_RA_AI"
                      IN3 := "DB_Scalling".RH_FD_Fan_Min,
                      IN4 := "DB_Scalling".RH_FD_Fan_Max,
                      Out13 => "DB102_ANALOG_DISPLAY".STAT9_RHFD_SPEED);
END_REGION

REGION Network 7: Speed LH Stoker | IW 200
   RUNG wire#powerrail
      "DB124_LH_STOKER_SPEED"(IN0 :=, IN1 :=, IN2 := "DB103_ANALOG_INPUT"."STAT13_Speed LH Stoker", IN3 := "DB_Scalling".LH_Stoker_Min, IN4 := "DB_Scalling".LH_Stoker_Max, IN5 :=, IN6 :=, IN7 :=, IN8 :=, IN9 :=, IN10 :=, IN11 :=, IN12 :=, IO19 :=, Out13 => "DB102_ANALOG_DISPLAY".STAT10_LHSTOKER_SPEED, Out14 =>, Out15 =>, Out16 =>, Out17 =>, Out18 =>)
   END_RUNG
   // the same network as SCL:
   "DB124_LH_STOKER_SPEED"(IN2 := "DB103_ANALOG_INPUT"."STAT13_Speed LH Stoker",   // "FB20_RA_AI"
                           IN3 := "DB_Scalling".LH_Stoker_Min,
                           IN4 := "DB_Scalling".LH_Stoker_Max,
                           Out13 => "DB102_ANALOG_DISPLAY".STAT10_LHSTOKER_SPEED);
END_REGION

REGION Network 8: Speed LH Stoker | IW 200
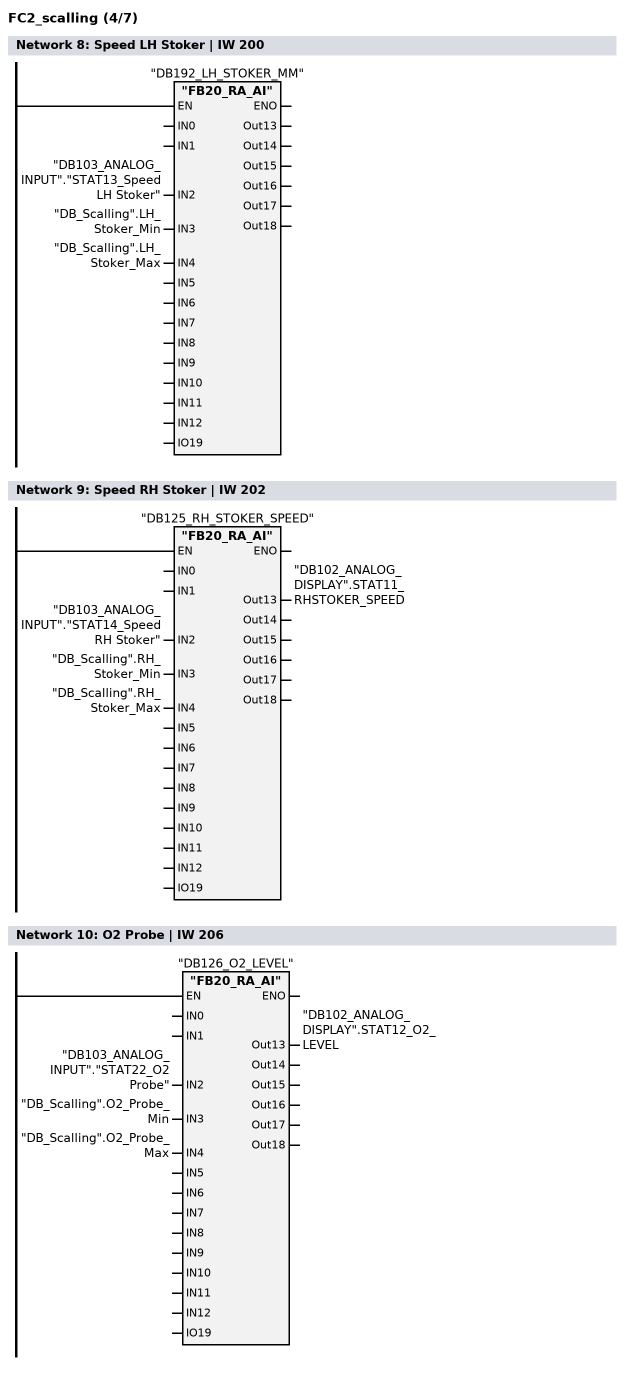
   RUNG wire#powerrail
      "DB192_LH_STOKER_MM"(IN0 :=, IN1 :=, IN2 := "DB103_ANALOG_INPUT"."STAT13_Speed LH Stoker", IN3 := "DB_Scalling".LH_Stoker_Min, IN4 := "DB_Scalling".LH_Stoker_Max, IN5 :=, IN6 :=, IN7 :=, IN8 :=, IN9 :=, IN10 :=, IN11 :=, IN12 :=, IO19 :=, Out13 =>, Out14 =>, Out15 =>, Out16 =>, Out17 =>, Out18 =>)
   END_RUNG
   // the same network as SCL:
   "DB192_LH_STOKER_MM"(IN2 := "DB103_ANALOG_INPUT"."STAT13_Speed LH Stoker",   // "FB20_RA_AI"
                        IN3 := "DB_Scalling".LH_Stoker_Min,
                        IN4 := "DB_Scalling".LH_Stoker_Max);
END_REGION

REGION Network 9: Speed RH Stoker | IW 202
   RUNG wire#powerrail
      "DB125_RH_STOKER_SPEED"(IN0 :=, IN1 :=, IN2 := "DB103_ANALOG_INPUT"."STAT14_Speed RH Stoker", IN3 := "DB_Scalling".RH_Stoker_Min, IN4 := "DB_Scalling".RH_Stoker_Max, IN5 :=, IN6 :=, IN7 :=, IN8 :=, IN9 :=, IN10 :=, IN11 :=, IN12 :=, IO19 :=, Out13 => "DB102_ANALOG_DISPLAY".STAT11_RHSTOKER_SPEED, Out14 =>, Out15 =>, Out16 =>, Out17 =>, Out18 =>)
   END_RUNG
   // the same network as SCL:
   "DB125_RH_STOKER_SPEED"(IN2 := "DB103_ANALOG_INPUT"."STAT14_Speed RH Stoker",   // "FB20_RA_AI"
                           IN3 := "DB_Scalling".RH_Stoker_Min,
                           IN4 := "DB_Scalling".RH_Stoker_Max,
                           Out13 => "DB102_ANALOG_DISPLAY".STAT11_RHSTOKER_SPEED);
END_REGION

REGION Network 10: O2 Probe | IW 206
   RUNG wire#powerrail
      "DB126_O2_LEVEL"(IN0 :=, IN1 :=, IN2 := "DB103_ANALOG_INPUT"."STAT22_O2 Probe", IN3 := "DB_Scalling".O2_Probe_Min, IN4 := "DB_Scalling".O2_Probe_Max, IN5 :=, IN6 :=, IN7 :=, IN8 :=, IN9 :=, IN10 :=, IN11 :=, IN12 :=, IO19 :=, Out13 => "DB102_ANALOG_DISPLAY".STAT12_O2_LEVEL, Out14 =>, Out15 =>, Out16 =>, Out17 =>, Out18 =>)
   END_RUNG
   // the same network as SCL:
   "DB126_O2_LEVEL"(IN2 := "DB103_ANALOG_INPUT"."STAT22_O2 Probe",   // "FB20_RA_AI"
                    IN3 := "DB_Scalling".O2_Probe_Min,
                    IN4 := "DB_Scalling".O2_Probe_Max,
                    Out13 => "DB102_ANALOG_DISPLAY".STAT12_O2_LEVEL);
END_REGION

REGION Network 11: MUL SUB O2 , CO2
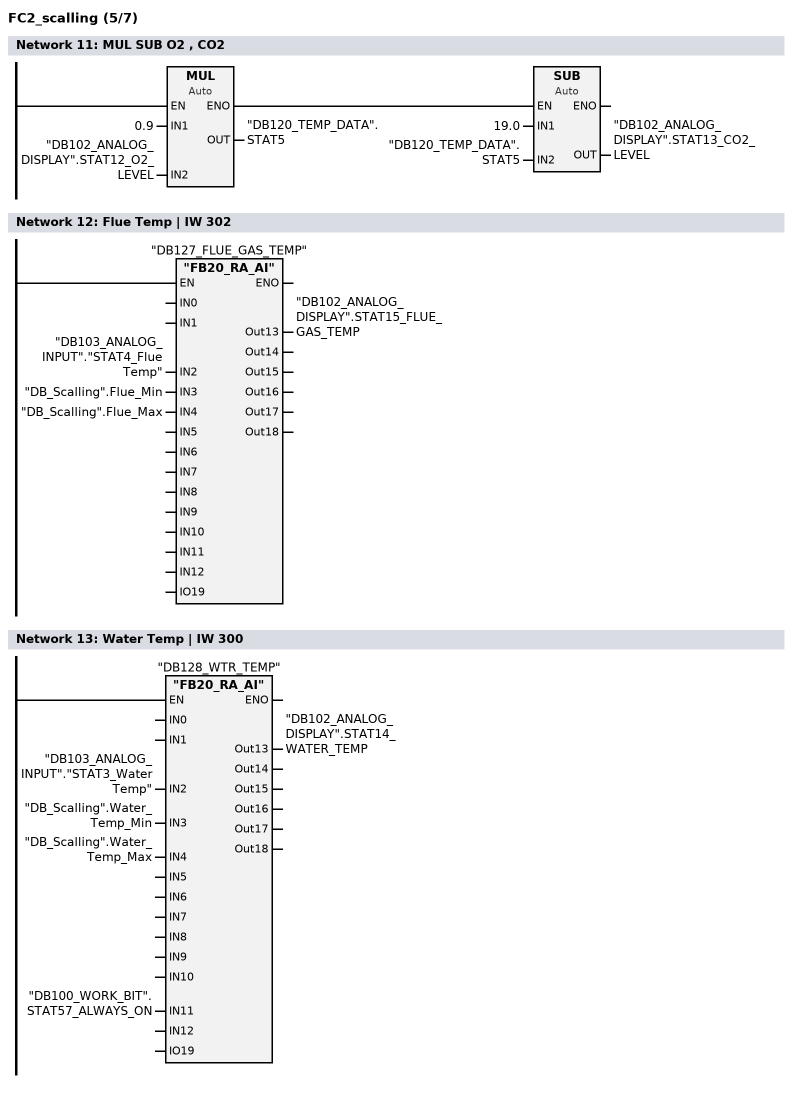
   RUNG wire#powerrail
      Mul(in1 := 0.9, in2 := "DB102_ANALOG_DISPLAY".STAT12_O2_LEVEL, out => "DB120_TEMP_DATA".STAT5)
      Sub(in1 := 19.0, in2 := "DB120_TEMP_DATA".STAT5, out => "DB102_ANALOG_DISPLAY".STAT13_CO2_LEVEL)
   END_RUNG
   // the same network as SCL:
   "DB120_TEMP_DATA".STAT5 := 0.9 * "DB102_ANALOG_DISPLAY".STAT12_O2_LEVEL;
   "DB102_ANALOG_DISPLAY".STAT13_CO2_LEVEL := 19.0 - "DB120_TEMP_DATA".STAT5;
END_REGION

REGION Network 12: Flue Temp | IW 302
   RUNG wire#powerrail
      "DB127_FLUE_GAS_TEMP"(IN0 :=, IN1 :=, IN2 := "DB103_ANALOG_INPUT"."STAT4_Flue Temp", IN3 := "DB_Scalling".Flue_Min, IN4 := "DB_Scalling".Flue_Max, IN5 :=, IN6 :=, IN7 :=, IN8 :=, IN9 :=, IN10 :=, IN11 :=, IN12 :=, IO19 :=, Out13 => "DB102_ANALOG_DISPLAY".STAT15_FLUE_GAS_TEMP, Out14 =>, Out15 =>, Out16 =>, Out17 =>, Out18 =>)
   END_RUNG
   // the same network as SCL:
   "DB127_FLUE_GAS_TEMP"(IN2 := "DB103_ANALOG_INPUT"."STAT4_Flue Temp",   // "FB20_RA_AI"
                         IN3 := "DB_Scalling".Flue_Min,
                         IN4 := "DB_Scalling".Flue_Max,
                         Out13 => "DB102_ANALOG_DISPLAY".STAT15_FLUE_GAS_TEMP);
END_REGION

REGION Network 13: Water Temp | IW 300
   RUNG wire#powerrail
      "DB128_WTR_TEMP"(IN0 :=, IN1 :=, IN2 := "DB103_ANALOG_INPUT"."STAT3_Water Temp", IN3 := "DB_Scalling".Water_Temp_Min, IN4 := "DB_Scalling".Water_Temp_Max, IN5 :=, IN6 :=, IN7 :=, IN8 :=, IN9 :=, IN10 :=, IN11 := "DB100_WORK_BIT".STAT57_ALWAYS_ON, IN12 :=, IO19 :=, Out13 => "DB102_ANALOG_DISPLAY".STAT14_WATER_TEMP, Out14 =>, Out15 =>, Out16 =>, Out17 =>, Out18 =>)
   END_RUNG
   // the same network as SCL:
   "DB128_WTR_TEMP"(IN2 := "DB103_ANALOG_INPUT"."STAT3_Water Temp",   // "FB20_RA_AI"
                    IN3 := "DB_Scalling".Water_Temp_Min,
                    IN4 := "DB_Scalling".Water_Temp_Max,
                    IN11 := "DB100_WORK_BIT".STAT57_ALWAYS_ON,
                    Out13 => "DB102_ANALOG_DISPLAY".STAT14_WATER_TEMP);
END_REGION

